LIN {X 0,Y 185.568,Z 561.36,A -85,B 0,C 180,E1 -22347.032,E2 -22347.032} C_VEL
LIN {X 0,Y 185.587,Z 561.366,A -85,B 0,C 180,E1 -22349.493,E2 -22349.493} C_VEL
LIN {X 0,Y 185.509,Z 561.379,A -85,B 0,C 180,E1 -22354.631,E2 -22354.631} C_VEL
LIN {X 0,Y 185.515,Z 561.377,A -85,B 0,C 180,E1 -22357.312,E2 -22357.312} C_VEL
LIN {X 0,Y 185.48,Z 561.382,A -85,B 0,C 180,E1 -22360.724,E2 -22360.724} C_VEL
LIN {X 0,Y 185.468,Z 561.376,A -85,B 0,C 180,E1 -22366.054,E2 -22366.054} C_VEL
LIN {X 0,Y 185.531,Z 561.532,A -85,B 0,C 180,E1 -22368.005,E2 -22368.005} C_VEL
LIN {X 0,Y 186.738,Z 566.432,A -85,B 0,C 180,E1 -22370.786,E2 -22370.786} C_VEL
LIN {X 0,Y 194.108,Z 583.862,A -85,B 0,C 180,E1 -22372.91,E2 -22372.91} C_VEL
LIN {X 0,Y 201.823,Z 604.433,A -85,B 0,C 180,E1 -22375.045,E2 -22375.045} C_VEL
LIN {X 0,Y 204.097,Z 623.143,A -85,B 0,C 180,E1 -22376.201,E2 -22376.201} C_VEL
LIN {X 0,Y 201.981,Z 663.7,A -85,B 0,C 180,E1 -22377.733,E2 -22377.733} C_VEL
LIN {X 0,Y 201.059,Z 669.51,A -85,B 0,C 180,E1 -22377.882,E2 -22377.882} C_VEL
LIN {X 0,Y 197.67,Z 678.837,A -85,B 0,C 180,E1 -22378.008,E2 -22378.008} C_VEL
LIN {X 0,Y 194.055,Z 688.023,A -85,B 0,C 180,E1 -22378.33,E2 -22378.33} C_VEL
LIN {X 0,Y 192.763,Z 693.612,A -85,B 0,C 180,E1 -22378.765,E2 -22378.765} C_VEL
LIN {X 0,Y 191.04,Z 704.06,A -85,B 0,C 180,E1 -22379.915,E2 -22379.915} C_VEL
LIN {X 0,Y 188.782,Z 716.056,A -85,B 0,C 180,E1 -22381.66,E2 -22381.66} C_VEL
LIN {X 0,Y 186.405,Z 726.819,A -85,B 0,C 180,E1 -22383.701,E2 -22383.701} C_VEL
LIN {X 0,Y 184.002,Z 736.963,A -85,B 0,C 180,E1 -22386.144,E2 -22386.144} C_VEL
LIN {X 0,Y 182.039,Z 744.915,A -85,B 0,C 180,E1 -22388.517,E2 -22388.517} C_VEL
LIN {X 0,Y 179.866,Z 753.724,A -85,B 0,C 180,E1 -22391.782,E2 -22391.782} C_VEL
LIN {X 0,Y 178.072,Z 760.784,A -85,B 0,C 180,E1 -22395.132,E2 -22395.132} C_VEL
LIN {X 0,Y 176.994,Z 766.43,A -85,B 0,C 180,E1 -22398.545,E2 -22398.545} C_VEL
LIN {X 0,Y 176.336,Z 770.82,A -85,B 0,C 180,E1 -22401.978,E2 -22401.978} C_VEL
LIN {X 0,Y 176.06,Z 774.084,A -85,B 0,C 180,E1 -22405.418,E2 -22405.418} C_VEL
LIN {X 0,Y 176.025,Z 775.685,A -85,B 0,C 180,E1 -22407.709,E2 -22407.709} C_VEL
LIN {X 0,Y 176.156,Z 776.867,A -85,B 0,C 180,E1 -22409.997,E2 -22409.997} C_VEL
LIN {X 0,Y 175.973,Z 777.736,A -85,B 0,C 180,E1 -22413.172,E2 -22413.172} C_VEL
LIN {X 0,Y 176.142,Z 777.8,A -85,B 0,C 180,E1 -22416.871,E2 -22416.871} C_VEL
LIN {X 0,Y 176.481,Z 777.341,A -85,B 0,C 180,E1 -22419.162,E2 -22419.162} C_VEL
LIN {X 0,Y 177.065,Z 776.47,A -85,B 0,C 180,E1 -22421.443,E2 -22421.443} C_VEL
LIN {X 0,Y 178.915,Z 773.51,A -85,B 0,C 180,E1 -22425.957,E2 -22425.957} C_VEL
LIN {X 0,Y 181.172,Z 770.182,A -85,B 0,C 180,E1 -22429.249,E2 -22429.249} C_VEL
LIN {X 0,Y 183.99,Z 765.836,A -85,B 0,C 180,E1 -22432.453,E2 -22432.453} C_VEL
LIN {X 0,Y 187.769,Z 759.389,A -85,B 0,C 180,E1 -22436.063,E2 -22436.063} C_VEL
LIN {X 0,Y 191.749,Z 752.298,A -85,B 0,C 180,E1 -22439.051,E2 -22439.051} C_VEL
LIN {X 0,Y 196.292,Z 743.558,A -85,B 0,C 180,E1 -22441.874,E2 -22441.874} C_VEL
LIN {X 0,Y 200.452,Z 734.678,A -85,B 0,C 180,E1 -22444.119,E2 -22444.119} C_VEL
LIN {X 0,Y 204.501,Z 725.05,A -85,B 0,C 180,E1 -22446.049,E2 -22446.049} C_VEL
LIN {X 0,Y 208.379,Z 714.565,A -85,B 0,C 180,E1 -22447.68,E2 -22447.68} C_VEL
LIN {X 0,Y 211.849,Z 703.058,A -85,B 0,C 180,E1 -22449.07,E2 -22449.07} C_VEL
LIN {X 0,Y 215.033,Z 690.143,A -85,B 0,C 180,E1 -22450.199,E2 -22450.199} C_VEL
LIN {X 0,Y 217.375,Z 677.531,A -85,B 0,C 180,E1 -22450.945,E2 -22450.945} C_VEL
LIN {X 0,Y 219.026,Z 660.991,A -85,B 0,C 180,E1 -22451.617,E2 -22451.617} C_VEL
LIN {X 0,Y 221.568,Z 630.722,A -85,B 0,C 180,E1 -22452.671,E2 -22452.671} C_VEL
LIN {X 0,Y 217.435,Z 619.879,A -85,B 0,C 180,E1 -22454.973,E2 -22454.973} C_VEL
LIN {X 0,Y 213.68,Z 611.836,A -85,B 0,C 180,E1 -22457.185,E2 -22457.185} C_VEL
LIN {X 0,Y 210.021,Z 604.877,A -85,B 0,C 180,E1 -22459.582,E2 -22459.582} C_VEL
LIN {X 0,Y 207.231,Z 599.872,A -85,B 0,C 180,E1 -22461.655,E2 -22461.655} C_VEL
LIN {X 0,Y 204.208,Z 594.895,A -85,B 0,C 180,E1 -22464.191,E2 -22464.191} C_VEL
LIN {X 0,Y 201.243,Z 589.954,A -85,B 0,C 180,E1 -22467.293,E2 -22467.293} C_VEL
LIN {X 0,Y 197.036,Z 583.326,A -85,B 0,C 180,E1 -22474.09,E2 -22474.09} C_VEL
LIN {X 0,Y 195.819,Z 581.983,A -85,B 0,C 180,E1 -22478.966,E2 -22478.966} C_VEL
LIN {X 0,Y 196.149,Z 581.812,A -85,B 0,C 180,E1 -22483.342,E2 -22483.342} C_VEL
LIN {X 0,Y 196.858,Z 582.371,A -85,B 0,C 180,E1 -22485.725,E2 -22485.725} C_VEL
LIN {X 0,Y 200.195,Z 586.287,A -85,B 0,C 180,E1 -22491.576,E2 -22491.576} C_VEL
LIN {X 0,Y 201.072,Z 587.621,A -85,B 0,C 180,E1 -22492.72,E2 -22492.72} C_VEL
LIN {X 0,Y 203.233,Z 590.314,A -85,B 0,C 180,E1 -22494.976,E2 -22494.976} C_VEL
LIN {X 0,Y 205.193,Z 592.528,A -85,B 0,C 180,E1 -22496.747,E2 -22496.747} C_VEL
LIN {X 0,Y 208.099,Z 597.214,A -85,B 0,C 180,E1 -22499.109,E2 -22499.109} C_VEL
LIN {X 0,Y 212.123,Z 603.731,A -85,B 0,C 180,E1 -22501.898,E2 -22501.898} C_VEL
LIN {X 0,Y 215.695,Z 610.557,A -85,B 0,C 180,E1 -22504.13,E2 -22504.13} C_VEL
LIN {X 0,Y 219.734,Z 618.887,A -85,B 0,C 180,E1 -22506.363,E2 -22506.363} C_VEL
LIN {X 0,Y 221.96,Z 624.2,A -85,B 0,C 180,E1 -22507.553,E2 -22507.553} C_VEL
LIN {X 0,Y 218.205,Z 667.202,A -85,B 0,C 180,E1 -22509.106,E2 -22509.106} C_VEL
LIN {X 0,Y 216.063,Z 680.58,A -85,B 0,C 180,E1 -22509.884,E2 -22509.884} C_VEL
LIN {X 0,Y 213.239,Z 693.467,A -85,B 0,C 180,E1 -22511.023,E2 -22511.023} C_VEL
LIN {X 0,Y 209.684,Z 705.782,A -85,B 0,C 180,E1 -22512.497,E2 -22512.497} C_VEL
LIN {X 0,Y 205.726,Z 717.054,A -85,B 0,C 180,E1 -22514.286,E2 -22514.286} C_VEL
LIN {X 0,Y 201.323,Z 727.735,A -85,B 0,C 180,E1 -22516.523,E2 -22516.523} C_VEL
LIN {X 0,Y 196.767,Z 737.303,A -85,B 0,C 180,E1 -22519.085,E2 -22519.085} C_VEL
LIN {X 0,Y 192.653,Z 744.988,A -85,B 0,C 180,E1 -22521.747,E2 -22521.747} C_VEL
LIN {X 0,Y 188.409,Z 752.132,A -85,B 0,C 180,E1 -22524.957,E2 -22524.957} C_VEL
LIN {X 0,Y 185.285,Z 757.04,A -85,B 0,C 180,E1 -22527.832,E2 -22527.832} C_VEL
LIN {X 0,Y 181.829,Z 762.034,A -85,B 0,C 180,E1 -22531.758,E2 -22531.758} C_VEL
LIN {X 0,Y 179.072,Z 765.618,A -85,B 0,C 180,E1 -22536.063,E2 -22536.063} C_VEL
LIN {X 0,Y 177.63,Z 767.253,A -85,B 0,C 180,E1 -22539.274,E2 -22539.274} C_VEL
LIN {X 0,Y 176.554,Z 768.081,A -85,B 0,C 180,E1 -22542.585,E2 -22542.585} C_VEL
LIN {X 0,Y 175.722,Z 767.804,A -85,B 0,C 180,E1 -22547.168,E2 -22547.168} C_VEL
LIN {X 0,Y 175.569,Z 766.792,A -85,B 0,C 180,E1 -22550.177,E2 -22550.177} C_VEL
LIN {X 0,Y 175.829,Z 763.978,A -85,B 0,C 180,E1 -22554.584,E2 -22554.584} C_VEL
LIN {X 0,Y 176.439,Z 760.818,A -85,B 0,C 180,E1 -22557.876,E2 -22557.876} C_VEL
LIN {X 0,Y 177.436,Z 755.952,A -85,B 0,C 180,E1 -22561.625,E2 -22561.625} C_VEL
LIN {X 0,Y 178.923,Z 749.619,A -85,B 0,C 180,E1 -22565.33,E2 -22565.33} C_VEL
LIN {X 0,Y 180.865,Z 741.806,A -85,B 0,C 180,E1 -22568.838,E2 -22568.838} C_VEL
LIN {X 0,Y 182.779,Z 734.376,A -85,B 0,C 180,E1 -22571.509,E2 -22571.509} C_VEL
LIN {X 0,Y 185.173,Z 724.662,A -85,B 0,C 180,E1 -22574.326,E2 -22574.326} C_VEL
LIN {X 0,Y 187.688,Z 713.78,A -85,B 0,C 180,E1 -22576.793,E2 -22576.793} C_VEL
LIN {X 0,Y 189.969,Z 702.456,A -85,B 0,C 180,E1 -22578.804,E2 -22578.804} C_VEL
LIN {X 0,Y 192.049,Z 690.439,A -85,B 0,C 180,E1 -22580.444,E2 -22580.444} C_VEL
LIN {X 0,Y 193.837,Z 676.765,A -85,B 0,C 180,E1 -22581.793,E2 -22581.793} C_VEL
LIN {X 0,Y 195.137,Z 663.168,A -85,B 0,C 180,E1 -22582.682,E2 -22582.682} C_VEL
LIN {X 0,Y 198.281,Z 606.848,A -85,B 0,C 180,E1 -22584.891,E2 -22584.891} C_VEL
LIN {X 0,Y 189.965,Z 584.27,A -85,B 0,C 180,E1 -22587.286,E2 -22587.286} C_VEL
LIN {X 0,Y 179.493,Z 563.052,A -85,B 0,C 180,E1 -22590.249,E2 -22590.249} C_VEL
LIN {X 0,Y 179.298,Z 562.148,A -85,B 0,C 180,E1 -22590.424,E2 -22590.424} C_VEL
LIN {X 0,Y 178.927,Z 562.19,A -85,B 0,C 180,E1 -22596.77,E2 -22596.77} C_VEL
LIN {X 0,Y 178.86,Z 562.199,A -85,B 0,C 180,E1 -22600.794,E2 -22600.794} C_VEL
LIN {X 0,Y 178.667,Z 562.228,A -85,B 0,C 180,E1 -22605.986,E2 -22605.986} C_VEL
LIN {X 0,Y 178.624,Z 562.227,A -85,B 0,C 180,E1 -22609.219,E2 -22609.219} C_VEL
LIN {X 0,Y 178.536,Z 562.233,A -85,B 0,C 180,E1 -22615.127,E2 -22615.127} C_VEL
LIN {X 0,Y 178.479,Z 562.25,A -85,B 0,C 180,E1 -22620.794,E2 -22620.794} C_VEL
LIN {X 0,Y 178.486,Z 562.25,A -85,B 0,C 180,E1 -22624.222,E2 -22624.222} C_VEL
LIN {X 0,Y 178.399,Z 562.257,A -85,B 0,C 180,E1 -22629.077,E2 -22629.077} C_VEL
LIN {X 0,Y 178.402,Z 562.255,A -85,B 0,C 180,E1 -22632.048,E2 -22632.048} C_VEL
LIN {X 0,Y 178.403,Z 562.263,A -85,B 0,C 180,E1 -22635.165,E2 -22635.165} C_VEL
LIN {X 0,Y 178.408,Z 562.255,A -85,B 0,C 180,E1 -22638.462,E2 -22638.462} C_VEL
LIN {X 0,Y 178.428,Z 562.257,A -85,B 0,C 180,E1 -22643.786,E2 -22643.786} C_VEL
LIN {X 0,Y 178.493,Z 562.25,A -85,B 0,C 180,E1 -22646.55,E2 -22646.55} C_VEL
LIN {X 0,Y 178.529,Z 562.232,A -85,B 0,C 180,E1 -22650.009,E2 -22650.009} C_VEL
LIN {X 0,Y 178.527,Z 562.242,A -85,B 0,C 180,E1 -22654.888,E2 -22654.888} C_VEL
LIN {X 0,Y 178.617,Z 562.226,A -85,B 0,C 180,E1 -22660.799,E2 -22660.799} C_VEL
LIN {X 0,Y 178.659,Z 562.228,A -85,B 0,C 180,E1 -22666.349,E2 -22666.349} C_VEL
LIN {X 0,Y 178.92,Z 562.192,A -85,B 0,C 180,E1 -22670.961,E2 -22670.961} C_VEL
LIN {X 0,Y 179.161,Z 562.167,A -85,B 0,C 180,E1 -22677.753,E2 -22677.753} C_VEL
LIN {X 0,Y 179.379,Z 562.14,A -85,B 0,C 180,E1 -22680.001,E2 -22680.001} C_VEL
LIN {X 0,Y 178.882,Z 562.19,A -85,B 0,C 180,E1 -22684.508,E2 -22684.508} C_VEL
LIN {X 0,Y 178.988,Z 562.189,A -85,B 0,C 180,E1 -22689.037,E2 -22689.037} C_VEL
LIN {X 0,Y 178.676,Z 562.217,A -85,B 0,C 180,E1 -22693.652,E2 -22693.652} C_VEL
LIN {X 0,Y 178.632,Z 562.232,A -85,B 0,C 180,E1 -22699.215,E2 -22699.215} C_VEL
LIN {X 0,Y 178.53,Z 562.217,A -85,B 0,C 180,E1 -22705.114,E2 -22705.114} C_VEL
LIN {X 0,Y 178.531,Z 562.247,A -85,B 0,C 180,E1 -22709.992,E2 -22709.992} C_VEL
LIN {X 0,Y 178.494,Z 562.254,A -85,B 0,C 180,E1 -22714.218,E2 -22714.218} C_VEL
LIN {X 0,Y 178.405,Z 562.262,A -85,B 0,C 180,E1 -22719.073,E2 -22719.073} C_VEL
LIN {X 0,Y 178.407,Z 562.261,A -85,B 0,C 180,E1 -22722.044,E2 -22722.044} C_VEL
LIN {X 0,Y 178.453,Z 562.293,A -85,B 0,C 180,E1 -22727.084,E2 -22727.084} C_VEL
LIN {X 0,Y 179.461,Z 566.426,A -85,B 0,C 180,E1 -22729.464,E2 -22729.464} C_VEL
LIN {X 0,Y 187.25,Z 584.258,A -85,B 0,C 180,E1 -22731.8,E2 -22731.8} C_VEL
LIN {X 0,Y 195.637,Z 606.702,A -85,B 0,C 180,E1 -22734.246,E2 -22734.246} C_VEL
LIN {X 0,Y 197.643,Z 623.334,A -85,B 0,C 180,E1 -22735.32,E2 -22735.32} C_VEL
LIN {X 0,Y 194.819,Z 675.043,A -85,B 0,C 180,E1 -22737.391,E2 -22737.391} C_VEL
LIN {X 0,Y 193.484,Z 687.523,A -85,B 0,C 180,E1 -22738.215,E2 -22738.215} C_VEL
LIN {X 0,Y 192.763,Z 693.612,A -85,B 0,C 180,E1 -22738.765,E2 -22738.765} C_VEL
LIN {X 0,Y 191.927,Z 697.302,A -85,B 0,C 180,E1 -22739.099,E2 -22739.099} C_VEL
LIN {X 0,Y 188.874,Z 704.35,A -85,B 0,C 180,E1 -22739.701,E2 -22739.701} C_VEL
LIN {X 0,Y 182.587,Z 716.046,A -85,B 0,C 180,E1 -22740.989,E2 -22740.989} C_VEL
LIN {X 0,Y 180.955,Z 721.015,A -85,B 0,C 180,E1 -22741.842,E2 -22741.842} C_VEL
LIN {X 0,Y 178.322,Z 732.128,A -85,B 0,C 180,E1 -22744.305,E2 -22744.305} C_VEL
LIN {X 0,Y 175.955,Z 741.248,A -85,B 0,C 180,E1 -22746.853,E2 -22746.853} C_VEL
LIN {X 0,Y 174.196,Z 748.419,A -85,B 0,C 180,E1 -22749.324,E2 -22749.324} C_VEL
LIN {X 0,Y 172.095,Z 756.546,A -85,B 0,C 180,E1 -22752.775,E2 -22752.775} C_VEL
LIN {X 0,Y 170.705,Z 762.018,A -85,B 0,C 180,E1 -22755.695,E2 -22755.695} C_VEL
LIN {X 0,Y 169.725,Z 767.371,A -85,B 0,C 180,E1 -22759.258,E2 -22759.258} C_VEL
LIN {X 0,Y 169.157,Z 771.486,A -85,B 0,C 180,E1 -22762.837,E2 -22762.837} C_VEL
LIN {X 0,Y 168.933,Z 774.775,A -85,B 0,C 180,E1 -22766.833,E2 -22766.833} C_VEL
LIN {X 0,Y 169.06,Z 776.481,A -85,B 0,C 180,E1 -22769.997,E2 -22769.997} C_VEL
LIN {X 0,Y 168.894,Z 777.381,A -85,B 0,C 180,E1 -22772.918,E2 -22772.918} C_VEL
LIN {X 0,Y 169.095,Z 777.617,A -85,B 0,C 180,E1 -22777.159,E2 -22777.159} C_VEL
LIN {X 0,Y 170.09,Z 776.42,A -85,B 0,C 180,E1 -22781.919,E2 -22781.919} C_VEL
LIN {X 0,Y 170.973,Z 775.213,A -85,B 0,C 180,E1 -22784.275,E2 -22784.275} C_VEL
LIN {X 0,Y 172.793,Z 772.668,A -85,B 0,C 180,E1 -22787.757,E2 -22787.757} C_VEL
LIN {X 0,Y 175.426,Z 769.138,A -85,B 0,C 180,E1 -22791.131,E2 -22791.131} C_VEL
LIN {X 0,Y 178.531,Z 764.559,A -85,B 0,C 180,E1 -22794.411,E2 -22794.411} C_VEL
LIN {X 0,Y 182.074,Z 758.817,A -85,B 0,C 180,E1 -22797.59,E2 -22797.59} C_VEL
LIN {X 0,Y 186.418,Z 751.681,A -85,B 0,C 180,E1 -22800.59,E2 -22800.59} C_VEL
LIN {X 0,Y 191.197,Z 742.922,A -85,B 0,C 180,E1 -22803.457,E2 -22803.457} C_VEL
LIN {X 0,Y 196.066,Z 733.037,A -85,B 0,C 180,E1 -22805.938,E2 -22805.938} C_VEL
LIN {X 0,Y 200.368,Z 723.04,A -85,B 0,C 180,E1 -22807.862,E2 -22807.862} C_VEL
LIN {X 0,Y 204.954,Z 710.562,A -85,B 0,C 180,E1 -22809.688,E2 -22809.688} C_VEL
LIN {X 0,Y 208.439,Z 698.994,A -85,B 0,C 180,E1 -22810.944,E2 -22810.944} C_VEL
LIN {X 0,Y 211.524,Z 685.589,A -85,B 0,C 180,E1 -22812.002,E2 -22812.002} C_VEL
LIN {X 0,Y 213.664,Z 672.766,A -85,B 0,C 180,E1 -22812.676,E2 -22812.676} C_VEL
LIN {X 0,Y 217.242,Z 633.882,A -85,B 0,C 180,E1 -22814.062,E2 -22814.062} C_VEL
LIN {X 0,Y 216.224,Z 630.484,A -85,B 0,C 180,E1 -22814.703,E2 -22814.703} C_VEL
LIN {X 0,Y 212.769,Z 621.671,A -85,B 0,C 180,E1 -22816.821,E2 -22816.821} C_VEL
LIN {X 0,Y 209.255,Z 614.22,A -85,B 0,C 180,E1 -22819.158,E2 -22819.158} C_VEL
LIN {X 0,Y 206.872,Z 609.624,A -85,B 0,C 180,E1 -22820.899,E2 -22820.899} C_VEL
LIN {X 0,Y 204.756,Z 605.627,A -85,B 0,C 180,E1 -22822.626,E2 -22822.626} C_VEL
LIN {X 0,Y 202.348,Z 601.388,A -85,B 0,C 180,E1 -22824.819,E2 -22824.819} C_VEL
LIN {X 0,Y 199.536,Z 596.507,A -85,B 0,C 180,E1 -22827.922,E2 -22827.922} C_VEL
LIN {X 0,Y 195.806,Z 590.238,A -85,B 0,C 180,E1 -22834.486,E2 -22834.486} C_VEL
LIN {X 0,Y 194.708,Z 588.892,A -85,B 0,C 180,E1 -22839.787,E2 -22839.787} C_VEL
LIN {X 0,Y 195.605,Z 589.104,A -85,B 0,C 180,E1 -22845.166,E2 -22845.166} C_VEL
LIN {X 0,Y 197.777,Z 592.058,A -85,B 0,C 180,E1 -22849.765,E2 -22849.765} C_VEL
LIN {X 0,Y 199.299,Z 593.862,A -85,B 0,C 180,E1 -22851.89,E2 -22851.89} C_VEL
LIN {X 0,Y 201.478,Z 596.956,A -85,B 0,C 180,E1 -22854.398,E2 -22854.398} C_VEL
LIN {X 0,Y 203.206,Z 598.85,A -85,B 0,C 180,E1 -22856.033,E2 -22856.033} C_VEL
LIN {X 0,Y 205.793,Z 603.268,A -85,B 0,C 180,E1 -22858.296,E2 -22858.296} C_VEL
LIN {X 0,Y 209.899,Z 610.214,A -85,B 0,C 180,E1 -22861.33,E2 -22861.33} C_VEL
LIN {X 0,Y 214.835,Z 620.382,A -85,B 0,C 180,E1 -22864.497,E2 -22864.497} C_VEL
LIN {X 0,Y 217.661,Z 627.045,A -85,B 0,C 180,E1 -22866.127,E2 -22866.127} C_VEL
LIN {X 0,Y 213.925,Z 667.397,A -85,B 0,C 180,E1 -22867.603,E2 -22867.603} C_VEL
LIN {X 0,Y 211.844,Z 679.957,A -85,B 0,C 180,E1 -22868.328,E2 -22868.328} C_VEL
LIN {X 0,Y 208.902,Z 692.992,A -85,B 0,C 180,E1 -22869.458,E2 -22869.458} C_VEL
LIN {X 0,Y 205.11,Z 705.704,A -85,B 0,C 180,E1 -22870.974,E2 -22870.974} C_VEL
LIN {X 0,Y 200.968,Z 717.062,A -85,B 0,C 180,E1 -22872.772,E2 -22872.772} C_VEL
LIN {X 0,Y 196.415,Z 727.596,A -85,B 0,C 180,E1 -22874.976,E2 -22874.976} C_VEL
LIN {X 0,Y 191.618,Z 737.127,A -85,B 0,C 180,E1 -22877.533,E2 -22877.533} C_VEL
LIN {X 0,Y 186.674,Z 745.816,A -85,B 0,C 180,E1 -22880.626,E2 -22880.626} C_VEL
LIN {X 0,Y 181.755,Z 753.527,A -85,B 0,C 180,E1 -22884.281,E2 -22884.281} C_VEL
LIN {X 0,Y 178.463,Z 758.249,A -85,B 0,C 180,E1 -22887.277,E2 -22887.277} C_VEL
LIN {X 0,Y 175.677,Z 761.951,A -85,B 0,C 180,E1 -22890.356,E2 -22890.356} C_VEL
LIN {X 0,Y 172.609,Z 765.631,A -85,B 0,C 180,E1 -22894.751,E2 -22894.751} C_VEL
LIN {X 0,Y 170.77,Z 767.512,A -85,B 0,C 180,E1 -22898.567,E2 -22898.567} C_VEL
LIN {X 0,Y 169.657,Z 768.284,A -85,B 0,C 180,E1 -22901.791,E2 -22901.791} C_VEL
LIN {X 0,Y 168.922,Z 768.289,A -85,B 0,C 180,E1 -22905.012,E2 -22905.012} C_VEL
LIN {X 0,Y 168.512,Z 767.446,A -85,B 0,C 180,E1 -22908.65,E2 -22908.65} C_VEL
LIN {X 0,Y 168.516,Z 765.591,A -85,B 0,C 180,E1 -22912.408,E2 -22912.408} C_VEL
LIN {X 0,Y 169.005,Z 762.581,A -85,B 0,C 180,E1 -22916.27,E2 -22916.27} C_VEL
LIN {X 0,Y 169.908,Z 758.132,A -85,B 0,C 180,E1 -22920.298,E2 -22920.298} C_VEL
LIN {X 0,Y 171.117,Z 752.906,A -85,B 0,C 180,E1 -22923.853,E2 -22923.853} C_VEL
LIN {X 0,Y 172.736,Z 746.503,A -85,B 0,C 180,E1 -22927.266,E2 -22927.266} C_VEL
LIN {X 0,Y 174.895,Z 738.452,A -85,B 0,C 180,E1 -22930.643,E2 -22930.643} C_VEL
LIN {X 0,Y 176.954,Z 730.378,A -85,B 0,C 180,E1 -22933.368,E2 -22933.368} C_VEL
LIN {X 0,Y 179.551,Z 720.14,A -85,B 0,C 180,E1 -22936.132,E2 -22936.132} C_VEL
LIN {X 0,Y 181.869,Z 709.949,A -85,B 0,C 180,E1 -22938.298,E2 -22938.298} C_VEL
LIN {X 0,Y 184.186,Z 698.043,A -85,B 0,C 180,E1 -22940.28,E2 -22940.28} C_VEL
LIN {X 0,Y 186.316,Z 685.283,A -85,B 0,C 180,E1 -22941.871,E2 -22941.871} C_VEL
LIN {X 0,Y 187.915,Z 671.4,A -85,B 0,C 180,E1 -22943.089,E2 -22943.089} C_VEL
LIN {X 0,Y 189.03,Z 658.7,A -85,B 0,C 180,E1 -22943.782,E2 -22943.782} C_VEL
LIN {X 0,Y 191.852,Z 608.295,A -85,B 0,C 180,E1 -22945.802,E2 -22945.802} C_VEL
LIN {X 0,Y 184.175,Z 587.474,A -85,B 0,C 180,E1 -22948.1,E2 -22948.1} C_VEL
LIN {X 0,Y 174.053,Z 566.979,A -85,B 0,C 180,E1 -22951.122,E2 -22951.122} C_VEL
LIN {X 0,Y 172.534,Z 564.575,A -85,B 0,C 180,E1 -22951.574,E2 -22951.574} C_VEL
LIN {X 0,Y 172.151,Z 563.038,A -85,B 0,C 180,E1 -22951.758,E2 -22951.758} C_VEL
LIN {X 0,Y 171.891,Z 563.068,A -85,B 0,C 180,E1 -22957.049,E2 -22957.049} C_VEL
LIN {X 0,Y 171.793,Z 563.078,A -85,B 0,C 180,E1 -22960.945,E2 -22960.945} C_VEL
LIN {X 0,Y 171.587,Z 563.112,A -85,B 0,C 180,E1 -22966.665,E2 -22966.665} C_VEL
LIN {X 0,Y 171.545,Z 563.107,A -85,B 0,C 180,E1 -22969.565,E2 -22969.565} C_VEL
LIN {X 0,Y 171.47,Z 563.117,A -85,B 0,C 180,E1 -22975.619,E2 -22975.619} C_VEL
LIN {X 0,Y 171.442,Z 563.128,A -85,B 0,C 180,E1 -22980.589,E2 -22980.589} C_VEL
LIN {X 0,Y 171.395,Z 563.135,A -85,B 0,C 180,E1 -22985.038,E2 -22985.038} C_VEL
LIN {X 0,Y 171.361,Z 563.135,A -85,B 0,C 180,E1 -22988.811,E2 -22988.811} C_VEL
LIN {X 0,Y 171.33,Z 563.142,A -85,B 0,C 180,E1 -22994.218,E2 -22994.218} C_VEL
LIN {X 0,Y 171.34,Z 563.13,A -85,B 0,C 180,E1 -22998.985,E2 -22998.985} C_VEL
LIN {X 0,Y 171.392,Z 563.125,A -85,B 0,C 180,E1 -23002.044,E2 -23002.044} C_VEL
LIN {X 0,Y 171.404,Z 563.133,A -85,B 0,C 180,E1 -23005.095,E2 -23005.095} C_VEL
LIN {X 0,Y 171.455,Z 563.111,A -85,B 0,C 180,E1 -23010.537,E2 -23010.537} C_VEL
LIN {X 0,Y 171.451,Z 563.128,A -85,B 0,C 180,E1 -23015.802,E2 -23015.802} C_VEL
LIN {X 0,Y 171.573,Z 563.101,A -85,B 0,C 180,E1 -23020.872,E2 -23020.872} C_VEL
LIN {X 0,Y 171.576,Z 563.107,A -85,B 0,C 180,E1 -23025.774,E2 -23025.774} C_VEL
LIN {X 0,Y 171.857,Z 563.072,A -85,B 0,C 180,E1 -23030.587,E2 -23030.587} C_VEL
LIN {X 0,Y 171.823,Z 563.07,A -85,B 0,C 180,E1 -23035.309,E2 -23035.309} C_VEL
LIN {X 0,Y 172.342,Z 563.016,A -85,B 0,C 180,E1 -23040.001,E2 -23040.001} C_VEL
LIN {X 0,Y 171.832,Z 563.068,A -85,B 0,C 180,E1 -23044.693,E2 -23044.693} C_VEL
LIN {X 0,Y 171.914,Z 563.071,A -85,B 0,C 180,E1 -23049.413,E2 -23049.413} C_VEL
LIN {X 0,Y 171.592,Z 563.103,A -85,B 0,C 180,E1 -23054.227,E2 -23054.227} C_VEL
LIN {X 0,Y 171.552,Z 563.111,A -85,B 0,C 180,E1 -23059.559,E2 -23059.559} C_VEL
LIN {X 0,Y 171.468,Z 563.099,A -85,B 0,C 180,E1 -23065.608,E2 -23065.608} C_VEL
LIN {X 0,Y 171.45,Z 563.127,A -85,B 0,C 180,E1 -23070.585,E2 -23070.585} C_VEL
LIN {X 0,Y 171.402,Z 563.135,A -85,B 0,C 180,E1 -23075.034,E2 -23075.034} C_VEL
LIN {X 0,Y 171.367,Z 563.139,A -85,B 0,C 180,E1 -23078.806,E2 -23078.806} C_VEL
LIN {X 0,Y 171.33,Z 563.141,A -85,B 0,C 180,E1 -23084.216,E2 -23084.216} C_VEL
LIN {X 0,Y 171.39,Z 563.23,A -85,B 0,C 180,E1 -23086.198,E2 -23086.198} C_VEL
LIN {X 0,Y 172.119,Z 566.116,A -85,B 0,C 180,E1 -23087.954,E2 -23087.954} C_VEL
LIN {X 0,Y 179.955,Z 583.631,A -85,B 0,C 180,E1 -23090.481,E2 -23090.481} C_VEL
LIN {X 0,Y 188.217,Z 605.357,A -85,B 0,C 180,E1 -23093.012,E2 -23093.012} C_VEL
LIN {X 0,Y 189.562,Z 609.48,A -85,B 0,C 180,E1 -23093.431,E2 -23093.431} C_VEL
LIN {X 0,Y 191.264,Z 624.539,A -85,B 0,C 180,E1 -23094.434,E2 -23094.434} C_VEL
LIN {X 0,Y 188.36,Z 675.155,A -85,B 0,C 180,E1 -23096.526,E2 -23096.526} C_VEL
LIN {X 0,Y 186.87,Z 688.248,A -85,B 0,C 180,E1 -23097.43,E2 -23097.43} C_VEL
LIN {X 0,Y 185.022,Z 700.485,A -85,B 0,C 180,E1 -23098.67,E2 -23098.67} C_VEL
LIN {X 0,Y 183.16,Z 710.788,A -85,B 0,C 180,E1 -23100.075,E2 -23100.075} C_VEL
LIN {X 0,Y 180.955,Z 721.015,A -85,B 0,C 180,E1 -23101.842,E2 -23101.842} C_VEL
LIN {X 0,Y 179.983,Z 724.29,A -85,B 0,C 180,E1 -23102.469,E2 -23102.469} C_VEL
LIN {X 0,Y 176.597,Z 730.43,A -85,B 0,C 180,E1 -23103.666,E2 -23103.666} C_VEL
LIN {X 0,Y 169.868,Z 740.256,A -85,B 0,C 180,E1 -23106.066,E2 -23106.066} C_VEL
LIN {X 0,Y 168.26,Z 744.347,A -85,B 0,C 180,E1 -23107.405,E2 -23107.405} C_VEL
LIN {X 0,Y 165.967,Z 752.979,A -85,B 0,C 180,E1 -23110.838,E2 -23110.838} C_VEL
LIN {X 0,Y 164.044,Z 760.117,A -85,B 0,C 180,E1 -23114.465,E2 -23114.465} C_VEL
LIN {X 0,Y 162.731,Z 766.632,A -85,B 0,C 180,E1 -23118.79,E2 -23118.79} C_VEL
LIN {X 0,Y 162.115,Z 770.872,A -85,B 0,C 180,E1 -23122.524,E2 -23122.524} C_VEL
LIN {X 0,Y 161.927,Z 773.093,A -85,B 0,C 180,E1 -23125.017,E2 -23125.017} C_VEL
LIN {X 0,Y 161.869,Z 774.804,A -85,B 0,C 180,E1 -23127.508,E2 -23127.508} C_VEL
LIN {X 0,Y 161.966,Z 776.09,A -85,B 0,C 180,E1 -23129.996,E2 -23129.996} C_VEL
LIN {X 0,Y 161.8,Z 776.951,A -85,B 0,C 180,E1 -23132.486,E2 -23132.486} C_VEL
LIN {X 0,Y 161.852,Z 777.407,A -85,B 0,C 180,E1 -23134.979,E2 -23134.979} C_VEL
LIN {X 0,Y 162.442,Z 777.08,A -85,B 0,C 180,E1 -23139.962,E2 -23139.962} C_VEL
LIN {X 0,Y 164.079,Z 775.243,A -85,B 0,C 180,E1 -23144.888,E2 -23144.888} C_VEL
LIN {X 0,Y 165.257,Z 773.706,A -85,B 0,C 180,E1 -23147.315,E2 -23147.315} C_VEL
LIN {X 0,Y 167.81,Z 770.634,A -85,B 0,C 180,E1 -23150.85,E2 -23150.85} C_VEL
LIN {X 0,Y 170.935,Z 766.544,A -85,B 0,C 180,E1 -23154.273,E2 -23154.273} C_VEL
LIN {X 0,Y 174.927,Z 760.807,A -85,B 0,C 180,E1 -23157.883,E2 -23157.883} C_VEL
LIN {X 0,Y 179.563,Z 753.708,A -85,B 0,C 180,E1 -23161.234,E2 -23161.234} C_VEL
LIN {X 0,Y 184.5,Z 745.501,A -85,B 0,C 180,E1 -23164.18,E2 -23164.18} C_VEL
LIN {X 0,Y 189.053,Z 737.153,A -85,B 0,C 180,E1 -23166.494,E2 -23166.494} C_VEL
LIN {X 0,Y 193.895,Z 726.981,A -85,B 0,C 180,E1 -23168.697,E2 -23168.697} C_VEL
LIN {X 0,Y 198.584,Z 715.696,A -85,B 0,C 180,E1 -23170.56,E2 -23170.56} C_VEL
LIN {X 0,Y 202.371,Z 704.743,A -85,B 0,C 180,E1 -23171.949,E2 -23171.949} C_VEL
LIN {X 0,Y 205.807,Z 692.559,A -85,B 0,C 180,E1 -23173.072,E2 -23173.072} C_VEL
LIN {X 0,Y 208.338,Z 680.87,A -85,B 0,C 180,E1 -23173.837,E2 -23173.837} C_VEL
LIN {X 0,Y 210.238,Z 666.915,A -85,B 0,C 180,E1 -23174.489,E2 -23174.489} C_VEL
LIN {X 0,Y 213.062,Z 636.036,A -85,B 0,C 180,E1 -23175.594,E2 -23175.594} C_VEL
LIN {X 0,Y 209.87,Z 627.208,A -85,B 0,C 180,E1 -23177.744,E2 -23177.744} C_VEL
LIN {X 0,Y 206.686,Z 620.131,A -85,B 0,C 180,E1 -23179.993,E2 -23179.993} C_VEL
LIN {X 0,Y 203.158,Z 612.726,A -85,B 0,C 180,E1 -23182.915,E2 -23182.915} C_VEL
LIN {X 0,Y 200.413,Z 607.725,A -85,B 0,C 180,E1 -23185.562,E2 -23185.562} C_VEL
LIN {X 0,Y 197.799,Z 602.988,A -85,B 0,C 180,E1 -23188.691,E2 -23188.691} C_VEL
LIN {X 0,Y 194.53,Z 597.085,A -85,B 0,C 180,E1 -23195.004,E2 -23195.004} C_VEL
LIN {X 0,Y 193.645,Z 595.824,A -85,B 0,C 180,E1 -23200.659,E2 -23200.659} C_VEL
LIN {X 0,Y 194.428,Z 596.053,A -85,B 0,C 180,E1 -23204.878,E2 -23204.878} C_VEL
LIN {X 0,Y 196.385,Z 598.879,A -85,B 0,C 180,E1 -23209.325,E2 -23209.325} C_VEL
LIN {X 0,Y 197.71,Z 600.414,A -85,B 0,C 180,E1 -23211.259,E2 -23211.259} C_VEL
LIN {X 0,Y 199.667,Z 603.486,A -85,B 0,C 180,E1 -23213.728,E2 -23213.728} C_VEL
LIN {X 0,Y 201.291,Z 605.224,A -85,B 0,C 180,E1 -23215.331,E2 -23215.331} C_VEL
LIN {X 0,Y 203.615,Z 609.484,A -85,B 0,C 180,E1 -23217.545,E2 -23217.545} C_VEL
LIN {X 0,Y 207.515,Z 616.508,A -85,B 0,C 180,E1 -23220.637,E2 -23220.637} C_VEL
LIN {X 0,Y 211.754,Z 625.735,A -85,B 0,C 180,E1 -23223.537,E2 -23223.537} C_VEL
LIN {X 0,Y 213.51,Z 630.019,A -85,B 0,C 180,E1 -23224.655,E2 -23224.655} C_VEL
LIN {X 0,Y 209.9,Z 667.334,A -85,B 0,C 180,E1 -23226.019,E2 -23226.019} C_VEL
LIN {X 0,Y 207.655,Z 680.352,A -85,B 0,C 180,E1 -23226.761,E2 -23226.761} C_VEL
LIN {X 0,Y 204.57,Z 693.413,A -85,B 0,C 180,E1 -23227.898,E2 -23227.898} C_VEL
LIN {X 0,Y 201.061,Z 704.804,A -85,B 0,C 180,E1 -23229.253,E2 -23229.253} C_VEL
LIN {X 0,Y 196.85,Z 715.9,A -85,B 0,C 180,E1 -23230.963,E2 -23230.963} C_VEL
LIN {X 0,Y 192.573,Z 725.607,A -85,B 0,C 180,E1 -23232.913,E2 -23232.913} C_VEL
LIN {X 0,Y 188.025,Z 734.495,A -85,B 0,C 180,E1 -23235.167,E2 -23235.167} C_VEL
LIN {X 0,Y 183.234,Z 742.781,A -85,B 0,C 180,E1 -23237.868,E2 -23237.868} C_VEL
LIN {X 0,Y 178.922,Z 749.524,A -85,B 0,C 180,E1 -23240.701,E2 -23240.701} C_VEL
LIN {X 0,Y 174.982,Z 755.066,A -85,B 0,C 180,E1 -23243.679,E2 -23243.679} C_VEL
LIN {X 0,Y 171.541,Z 759.52,A -85,B 0,C 180,E1 -23246.785,E2 -23246.785} C_VEL
LIN {X 0,Y 167.674,Z 764.132,A -85,B 0,C 180,E1 -23251.269,E2 -23251.269} C_VEL
LIN {X 0,Y 166.266,Z 765.645,A -85,B 0,C 180,E1 -23253.332,E2 -23253.332} C_VEL
LIN {X 0,Y 164.37,Z 767.418,A -85,B 0,C 180,E1 -23256.768,E2 -23256.768} C_VEL
LIN {X 0,Y 162.979,Z 768.386,A -85,B 0,C 180,E1 -23260.301,E2 -23260.301} C_VEL
LIN {X 0,Y 162.004,Z 768.543,A -85,B 0,C 180,E1 -23263.954,E2 -23263.954} C_VEL
LIN {X 0,Y 161.462,Z 767.818,A -85,B 0,C 180,E1 -23267.726,E2 -23267.726} C_VEL
LIN {X 0,Y 161.418,Z 765.6,A -85,B 0,C 180,E1 -23272.448,E2 -23272.448} C_VEL
LIN {X 0,Y 162.068,Z 761.844,A -85,B 0,C 180,E1 -23277.181,E2 -23277.181} C_VEL
LIN {X 0,Y 162.906,Z 757.83,A -85,B 0,C 180,E1 -23280.763,E2 -23280.763} C_VEL
LIN {X 0,Y 164.307,Z 752.072,A -85,B 0,C 180,E1 -23284.68,E2 -23284.68} C_VEL
LIN {X 0,Y 166.192,Z 744.867,A -85,B 0,C 180,E1 -23288.485,E2 -23288.485} C_VEL
LIN {X 0,Y 168.356,Z 737.151,A -85,B 0,C 180,E1 -23291.702,E2 -23291.702} C_VEL
LIN {X 0,Y 170.842,Z 727.796,A -85,B 0,C 180,E1 -23294.8,E2 -23294.8} C_VEL
LIN {X 0,Y 173.651,Z 716.703,A -85,B 0,C 180,E1 -23297.669,E2 -23297.669} C_VEL
LIN {X 0,Y 176.228,Z 705.286,A -85,B 0,C 180,E1 -23299.955,E2 -23299.955} C_VEL
LIN {X 0,Y 178.706,Z 692.119,A -85,B 0,C 180,E1 -23301.949,E2 -23301.949} C_VEL
LIN {X 0,Y 180.566,Z 679.605,A -85,B 0,C 180,E1 -23303.333,E2 -23303.333} C_VEL
LIN {X 0,Y 182.015,Z 666.866,A -85,B 0,C 180,E1 -23304.291,E2 -23304.291} C_VEL
LIN {X 0,Y 183.522,Z 643.161,A -85,B 0,C 180,E1 -23305.363,E2 -23305.363} C_VEL
LIN {X 0,Y 185.417,Z 609.703,A -85,B 0,C 180,E1 -23306.752,E2 -23306.752} C_VEL
LIN {X 0,Y 178.628,Z 591.12,A -85,B 0,C 180,E1 -23308.905,E2 -23308.905} C_VEL
LIN {X 0,Y 168.975,Z 571.456,A -85,B 0,C 180,E1 -23311.92,E2 -23311.92} C_VEL
LIN {X 0,Y 165.178,Z 565.112,A -85,B 0,C 180,E1 -23313.128,E2 -23313.128} C_VEL
LIN {X 0,Y 164.908,Z 563.942,A -85,B 0,C 180,E1 -23313.363,E2 -23313.363} C_VEL
LIN {X 0,Y 164.853,Z 563.946,A -85,B 0,C 180,E1 -23317.351,E2 -23317.351} C_VEL
LIN {X 0,Y 164.744,Z 563.953,A -85,B 0,C 180,E1 -23321.139,E2 -23321.139} C_VEL
LIN {X 0,Y 164.507,Z 563.994,A -85,B 0,C 180,E1 -23327.404,E2 -23327.404} C_VEL
LIN {X 0,Y 164.474,Z 563.981,A -85,B 0,C 180,E1 -23329.993,E2 -23329.993} C_VEL
LIN {X 0,Y 164.394,Z 564.003,A -85,B 0,C 180,E1 -23336.137,E2 -23336.137} C_VEL
LIN {X 0,Y 164.376,Z 564.003,A -85,B 0,C 180,E1 -23341.23,E2 -23341.23} C_VEL
LIN {X 0,Y 164.297,Z 564.021,A -85,B 0,C 180,E1 -23346.793,E2 -23346.793} C_VEL
LIN {X 0,Y 164.294,Z 564.008,A -85,B 0,C 180,E1 -23349.919,E2 -23349.919} C_VEL
LIN {X 0,Y 164.283,Z 564.017,A -85,B 0,C 180,E1 -23353.345,E2 -23353.345} C_VEL
LIN {X 0,Y 164.297,Z 564.019,A -85,B 0,C 180,E1 -23356.812,E2 -23356.812} C_VEL
LIN {X 0,Y 164.3,Z 564,A -85,B 0,C 180,E1 -23360.355,E2 -23360.355} C_VEL
LIN {X 0,Y 164.336,Z 564.013,A -85,B 0,C 180,E1 -23364.352,E2 -23364.352} C_VEL
LIN {X 0,Y 164.397,Z 563.997,A -85,B 0,C 180,E1 -23369.138,E2 -23369.138} C_VEL
LIN {X 0,Y 164.413,Z 564,A -85,B 0,C 180,E1 -23374.695,E2 -23374.695} C_VEL
LIN {X 0,Y 164.47,Z 563.988,A -85,B 0,C 180,E1 -23380.074,E2 -23380.074} C_VEL
LIN {X 0,Y 164.506,Z 563.984,A -85,B 0,C 180,E1 -23385.149,E2 -23385.149} C_VEL
LIN {X 0,Y 164.777,Z 563.955,A -85,B 0,C 180,E1 -23390.178,E2 -23390.178} C_VEL
LIN {X 0,Y 164.84,Z 563.936,A -85,B 0,C 180,E1 -23392.653,E2 -23392.653} C_VEL
LIN {X 0,Y 165.056,Z 563.922,A -85,B 0,C 180,E1 -23397.561,E2 -23397.561} C_VEL
LIN {X 0,Y 165.304,Z 563.893,A -85,B 0,C 180,E1 -23400.001,E2 -23400.001} C_VEL
LIN {X 0,Y 164.87,Z 563.946,A -85,B 0,C 180,E1 -23407.348,E2 -23407.348} C_VEL
LIN {X 0,Y 164.76,Z 563.958,A -85,B 0,C 180,E1 -23411.146,E2 -23411.146} C_VEL
LIN {X 0,Y 164.494,Z 563.997,A -85,B 0,C 180,E1 -23417.403,E2 -23417.403} C_VEL
LIN {X 0,Y 164.483,Z 563.987,A -85,B 0,C 180,E1 -23419.989,E2 -23419.989} C_VEL
LIN {X 0,Y 164.395,Z 563.985,A -85,B 0,C 180,E1 -23426.127,E2 -23426.127} C_VEL
LIN {X 0,Y 164.384,Z 564.006,A -85,B 0,C 180,E1 -23431.226,E2 -23431.226} C_VEL
LIN {X 0,Y 164.304,Z 564.019,A -85,B 0,C 180,E1 -23436.788,E2 -23436.788} C_VEL
LIN {X 0,Y 164.3,Z 564.018,A -85,B 0,C 180,E1 -23439.915,E2 -23439.915} C_VEL
LIN {X 0,Y 164.299,Z 564.093,A -85,B 0,C 180,E1 -23445.22,E2 -23445.22} C_VEL
LIN {X 0,Y 164.773,Z 566.021,A -85,B 0,C 180,E1 -23446.367,E2 -23446.367} C_VEL
LIN {X 0,Y 172.1,Z 581.703,A -85,B 0,C 180,E1 -23448.838,E2 -23448.838} C_VEL
LIN {X 0,Y 178.399,Z 597.553,A -85,B 0,C 180,E1 -23450.936,E2 -23450.936} C_VEL
LIN {X 0,Y 183.381,Z 611.315,A -85,B 0,C 180,E1 -23452.524,E2 -23452.524} C_VEL
LIN {X 0,Y 184.92,Z 625.31,A -85,B 0,C 180,E1 -23453.486,E2 -23453.486} C_VEL
LIN {X 0,Y 181.95,Z 674.923,A -85,B 0,C 180,E1 -23455.601,E2 -23455.601} C_VEL
LIN {X 0,Y 180.404,Z 687.987,A -85,B 0,C 180,E1 -23456.528,E2 -23456.528} C_VEL
LIN {X 0,Y 178.582,Z 699.662,A -85,B 0,C 180,E1 -23457.738,E2 -23457.738} C_VEL
LIN {X 0,Y 176.665,Z 710.09,A -85,B 0,C 180,E1 -23459.187,E2 -23459.187} C_VEL
LIN {X 0,Y 174.002,Z 722.001,A -85,B 0,C 180,E1 -23461.335,E2 -23461.335} C_VEL
LIN {X 0,Y 171.39,Z 732.692,A -85,B 0,C 180,E1 -23463.841,E2 -23463.841} C_VEL
LIN {X 0,Y 168.812,Z 741.869,A -85,B 0,C 180,E1 -23466.54,E2 -23466.54} C_VEL
LIN {X 0,Y 168.26,Z 744.347,A -85,B 0,C 180,E1 -23467.405,E2 -23467.405} C_VEL
LIN {X 0,Y 167.369,Z 746.996,A -85,B 0,C 180,E1 -23468.358,E2 -23468.358} C_VEL
LIN {X 0,Y 165.085,Z 750.683,A -85,B 0,C 180,E1 -23469.757,E2 -23469.757} C_VEL
LIN {X 0,Y 158.586,Z 758.209,A -85,B 0,C 180,E1 -23473.238,E2 -23473.238} C_VEL
LIN {X 0,Y 156.764,Z 761.191,A -85,B 0,C 180,E1 -23474.98,E2 -23474.98} C_VEL
LIN {X 0,Y 156.47,Z 762.168,A -85,B 0,C 180,E1 -23475.597,E2 -23475.597} C_VEL
LIN {X 0,Y 155.452,Z 767.498,A -85,B 0,C 180,E1 -23479.578,E2 -23479.578} C_VEL
LIN {X 0,Y 154.909,Z 771.472,A -85,B 0,C 180,E1 -23483.484,E2 -23483.484} C_VEL
LIN {X 0,Y 154.779,Z 774.354,A -85,B 0,C 180,E1 -23487.394,E2 -23487.394} C_VEL
LIN {X 0,Y 154.874,Z 775.692,A -85,B 0,C 180,E1 -23489.996,E2 -23489.996} C_VEL
LIN {X 0,Y 154.719,Z 776.603,A -85,B 0,C 180,E1 -23492.6,E2 -23492.6} C_VEL
LIN {X 0,Y 154.761,Z 777.126,A -85,B 0,C 180,E1 -23495.207,E2 -23495.207} C_VEL
LIN {X 0,Y 154.971,Z 777.25,A -85,B 0,C 180,E1 -23497.816,E2 -23497.816} C_VEL
LIN {X 0,Y 156.186,Z 776.284,A -85,B 0,C 180,E1 -23502.998,E2 -23502.998} C_VEL
LIN {X 0,Y 158.476,Z 773.8,A -85,B 0,C 180,E1 -23508.081,E2 -23508.081} C_VEL
LIN {X 0,Y 161.195,Z 770.842,A -85,B 0,C 180,E1 -23511.748,E2 -23511.748} C_VEL
LIN {X 0,Y 164.48,Z 766.898,A -85,B 0,C 180,E1 -23515.291,E2 -23515.291} C_VEL
LIN {X 0,Y 168.59,Z 761.53,A -85,B 0,C 180,E1 -23518.902,E2 -23518.902} C_VEL
LIN {X 0,Y 173.585,Z 754.435,A -85,B 0,C 180,E1 -23522.439,E2 -23522.439} C_VEL
LIN {X 0,Y 178.729,Z 746.452,A -85,B 0,C 180,E1 -23525.446,E2 -23525.446} C_VEL
LIN {X 0,Y 184.451,Z 736.615,A -85,B 0,C 180,E1 -23528.251,E2 -23528.251} C_VEL
LIN {X 0,Y 189.037,Z 727.541,A -85,B 0,C 180,E1 -23530.234,E2 -23530.234} C_VEL
LIN {X 0,Y 193.901,Z 716.412,A -85,B 0,C 180,E1 -23532.104,E2 -23532.104} C_VEL
LIN {X 0,Y 197.846,Z 705.656,A -85,B 0,C 180,E1 -23533.487,E2 -23533.487} C_VEL
LIN {X 0,Y 201.558,Z 693.267,A -85,B 0,C 180,E1 -23534.663,E2 -23534.663} C_VEL
LIN {X 0,Y 204.334,Z 681.114,A -85,B 0,C 180,E1 -23535.462,E2 -23535.462} C_VEL
LIN {X 0,Y 206.3,Z 667.72,A -85,B 0,C 180,E1 -23536.1,E2 -23536.1} C_VEL
LIN {X 0,Y 209.096,Z 638.868,A -85,B 0,C 180,E1 -23537.148,E2 -23537.148} C_VEL
LIN {X 0,Y 206.519,Z 631.443,A -85,B 0,C 180,E1 -23539.066,E2 -23539.066} C_VEL
LIN {X 0,Y 203.569,Z 624.557,A -85,B 0,C 180,E1 -23541.407,E2 -23541.407} C_VEL
LIN {X 0,Y 200.539,Z 618.09,A -85,B 0,C 180,E1 -23544.144,E2 -23544.144} C_VEL
LIN {X 0,Y 198.456,Z 613.985,A -85,B 0,C 180,E1 -23546.378,E2 -23546.378} C_VEL
LIN {X 0,Y 196.209,Z 609.588,A -85,B 0,C 180,E1 -23549.325,E2 -23549.325} C_VEL
LIN {X 0,Y 193.336,Z 604.018,A -85,B 0,C 180,E1 -23555.329,E2 -23555.329} C_VEL
LIN {X 0,Y 192.594,Z 602.816,A -85,B 0,C 180,E1 -23560.826,E2 -23560.826} C_VEL
LIN {X 0,Y 193.307,Z 603.168,A -85,B 0,C 180,E1 -23564.788,E2 -23564.788} C_VEL
LIN {X 0,Y 196.079,Z 606.852,A -85,B 0,C 180,E1 -23570.516,E2 -23570.516} C_VEL
LIN {X 0,Y 198.124,Z 610.248,A -85,B 0,C 180,E1 -23573.304,E2 -23573.304} C_VEL
LIN {X 0,Y 199.528,Z 611.846,A -85,B 0,C 180,E1 -23574.753,E2 -23574.753} C_VEL
LIN {X 0,Y 201.628,Z 616.015,A -85,B 0,C 180,E1 -23576.921,E2 -23576.921} C_VEL
LIN {X 0,Y 204.968,Z 622.229,A -85,B 0,C 180,E1 -23579.714,E2 -23579.714} C_VEL
LIN {X 0,Y 209.164,Z 631.994,A -85,B 0,C 180,E1 -23582.819,E2 -23582.819} C_VEL
LIN {X 0,Y 209.593,Z 633.135,A -85,B 0,C 180,E1 -23583.121,E2 -23583.121} C_VEL
LIN {X 0,Y 206.032,Z 667.573,A -85,B 0,C 180,E1 -23584.374,E2 -23584.374} C_VEL
LIN {X 0,Y 203.633,Z 680.903,A -85,B 0,C 180,E1 -23585.144,E2 -23585.144} C_VEL
LIN {X 0,Y 200.409,Z 693.828,A -85,B 0,C 180,E1 -23586.275,E2 -23586.275} C_VEL
LIN {X 0,Y 196.332,Z 706.364,A -85,B 0,C 180,E1 -23587.788,E2 -23587.788} C_VEL
LIN {X 0,Y 191.831,Z 717.506,A -85,B 0,C 180,E1 -23589.555,E2 -23589.555} C_VEL
LIN {X 0,Y 186.682,Z 728.237,A -85,B 0,C 180,E1 -23591.83,E2 -23591.83} C_VEL
LIN {X 0,Y 181.406,Z 737.659,A -85,B 0,C 180,E1 -23594.423,E2 -23594.423} C_VEL
LIN {X 0,Y 176.522,Z 745.309,A -85,B 0,C 180,E1 -23597.164,E2 -23597.164} C_VEL
LIN {X 0,Y 172.112,Z 751.624,A -85,B 0,C 180,E1 -23600.097,E2 -23600.097} C_VEL
LIN {X 0,Y 168.11,Z 756.745,A -85,B 0,C 180,E1 -23603.123,E2 -23603.123} C_VEL
LIN {X 0,Y 163.533,Z 762.019,A -85,B 0,C 180,E1 -23607.418,E2 -23607.418} C_VEL
LIN {X 0,Y 160.04,Z 765.635,A -85,B 0,C 180,E1 -23611.799,E2 -23611.799} C_VEL
LIN {X 0,Y 157.322,Z 767.914,A -85,B 0,C 180,E1 -23616.482,E2 -23616.482} C_VEL
LIN {X 0,Y 155.938,Z 768.703,A -85,B 0,C 180,E1 -23619.995,E2 -23619.995} C_VEL
LIN {X 0,Y 155.003,Z 768.738,A -85,B 0,C 180,E1 -23623.499,E2 -23623.499} C_VEL
LIN {X 0,Y 154.421,Z 768.102,A -85,B 0,C 180,E1 -23626.952,E2 -23626.952} C_VEL
LIN {X 0,Y 154.247,Z 766.583,A -85,B 0,C 180,E1 -23630.764,E2 -23630.764} C_VEL
LIN {X 0,Y 154.564,Z 763.892,A -85,B 0,C 180,E1 -23634.928,E2 -23634.928} C_VEL
LIN {X 0,Y 155.418,Z 759.873,A -85,B 0,C 180,E1 -23639.222,E2 -23639.222} C_VEL
LIN {X 0,Y 156.755,Z 754.119,A -85,B 0,C 180,E1 -23643.723,E2 -23643.723} C_VEL
LIN {X 0,Y 158.408,Z 747.948,A -85,B 0,C 180,E1 -23647.433,E2 -23647.433} C_VEL
LIN {X 0,Y 160.389,Z 740.872,A -85,B 0,C 180,E1 -23650.818,E2 -23650.818} C_VEL
LIN {X 0,Y 163.07,Z 731.399,A -85,B 0,C 180,E1 -23654.377,E2 -23654.377} C_VEL
LIN {X 0,Y 165.893,Z 720.959,A -85,B 0,C 180,E1 -23657.442,E2 -23657.442} C_VEL
LIN {X 0,Y 168.456,Z 710.731,A -85,B 0,C 180,E1 -23659.79,E2 -23659.79} C_VEL
LIN {X 0,Y 171.036,Z 698.38,A -85,B 0,C 180,E1 -23661.99,E2 -23661.99} C_VEL
LIN {X 0,Y 173.232,Z 686.298,A -85,B 0,C 180,E1 -23663.598,E2 -23663.598} C_VEL
LIN {X 0,Y 174.907,Z 672.825,A -85,B 0,C 180,E1 -23664.889,E2 -23664.889} C_VEL
LIN {X 0,Y 176.113,Z 660.59,A -85,B 0,C 180,E1 -23665.628,E2 -23665.628} C_VEL
LIN {X 0,Y 179.207,Z 611.63,A -85,B 0,C 180,E1 -23667.706,E2 -23667.706} C_VEL
LIN {X 0,Y 173.065,Z 594.633,A -85,B 0,C 180,E1 -23669.773,E2 -23669.773} C_VEL
LIN {X 0,Y 163.863,Z 575.789,A -85,B 0,C 180,E1 -23672.781,E2 -23672.781} C_VEL
LIN {X 0,Y 159.411,Z 568.526,A -85,B 0,C 180,E1 -23674.271,E2 -23674.271} C_VEL
LIN {X 0,Y 157.979,Z 565.957,A -85,B 0,C 180,E1 -23674.789,E2 -23674.789} C_VEL
LIN {X 0,Y 157.738,Z 564.824,A -85,B 0,C 180,E1 -23674.956,E2 -23674.956} C_VEL
LIN {X 0,Y 157.812,Z 564.826,A -85,B 0,C 180,E1 -23677.681,E2 -23677.681} C_VEL
LIN {X 0,Y 157.675,Z 564.831,A -85,B 0,C 180,E1 -23681.312,E2 -23681.312} C_VEL
LIN {X 0,Y 157.479,Z 564.865,A -85,B 0,C 180,E1 -23685.535,E2 -23685.535} C_VEL
LIN {X 0,Y 157.371,Z 564.855,A -85,B 0,C 180,E1 -23690.936,E2 -23690.936} C_VEL
LIN {X 0,Y 157.316,Z 564.886,A -85,B 0,C 180,E1 -23696.688,E2 -23696.688} C_VEL
LIN {X 0,Y 157.277,Z 564.883,A -85,B 0,C 180,E1 -23702.431,E2 -23702.431} C_VEL
LIN {X 0,Y 157.271,Z 564.896,A -85,B 0,C 180,E1 -23706.453,E2 -23706.453} C_VEL
LIN {X 0,Y 157.214,Z 564.892,A -85,B 0,C 180,E1 -23712.114,E2 -23712.114} C_VEL
LIN {X 0,Y 157.215,Z 564.895,A -85,B 0,C 180,E1 -23717.893,E2 -23717.893} C_VEL
LIN {X 0,Y 157.273,Z 564.889,A -85,B 0,C 180,E1 -23723.554,E2 -23723.554} C_VEL
LIN {X 0,Y 157.3,Z 564.885,A -85,B 0,C 180,E1 -23728.099,E2 -23728.099} C_VEL
LIN {X 0,Y 157.322,Z 564.876,A -85,B 0,C 180,E1 -23733.468,E2 -23733.468} C_VEL
LIN {X 0,Y 157.398,Z 564.871,A -85,B 0,C 180,E1 -23739.673,E2 -23739.673} C_VEL
LIN {X 0,Y 157.442,Z 564.86,A -85,B 0,C 180,E1 -23744.466,E2 -23744.466} C_VEL
LIN {X 0,Y 157.698,Z 564.838,A -85,B 0,C 180,E1 -23749.733,E2 -23749.733} C_VEL
LIN {X 0,Y 157.776,Z 564.816,A -85,B 0,C 180,E1 -23752.322,E2 -23752.322} C_VEL
LIN {X 0,Y 158.267,Z 564.769,A -85,B 0,C 180,E1 -23760.001,E2 -23760.001} C_VEL
LIN {X 0,Y 157.83,Z 564.824,A -85,B 0,C 180,E1 -23767.678,E2 -23767.678} C_VEL
LIN {X 0,Y 157.689,Z 564.836,A -85,B 0,C 180,E1 -23771.314,E2 -23771.314} C_VEL
LIN {X 0,Y 157.466,Z 564.869,A -85,B 0,C 180,E1 -23775.534,E2 -23775.534} C_VEL
LIN {X 0,Y 157.378,Z 564.864,A -85,B 0,C 180,E1 -23780.933,E2 -23780.933} C_VEL
LIN {X 0,Y 157.319,Z 564.869,A -85,B 0,C 180,E1 -23786.68,E2 -23786.68} C_VEL
LIN {X 0,Y 157.285,Z 564.889,A -85,B 0,C 180,E1 -23792.427,E2 -23792.427} C_VEL
LIN {X 0,Y 157.277,Z 564.893,A -85,B 0,C 180,E1 -23796.448,E2 -23796.448} C_VEL
LIN {X 0,Y 157.202,Z 564.902,A -85,B 0,C 180,E1 -23802.115,E2 -23802.115} C_VEL
LIN {X 0,Y 157.247,Z 564.92,A -85,B 0,C 180,E1 -23804.127,E2 -23804.127} C_VEL
LIN {X 0,Y 157.35,Z 565.557,A -85,B 0,C 180,E1 -23804.562,E2 -23804.562} C_VEL
LIN {X 0,Y 159.21,Z 569.422,A -85,B 0,C 180,E1 -23805.271,E2 -23805.271} C_VEL
LIN {X 0,Y 166.506,Z 585.06,A -85,B 0,C 180,E1 -23807.883,E2 -23807.883} C_VEL
LIN {X 0,Y 172.549,Z 600.27,A -85,B 0,C 180,E1 -23809.973,E2 -23809.973} C_VEL
LIN {X 0,Y 177.322,Z 614.138,A -85,B 0,C 180,E1 -23811.626,E2 -23811.626} C_VEL
LIN {X 0,Y 178.603,Z 626.134,A -85,B 0,C 180,E1 -23812.487,E2 -23812.487} C_VEL
LIN {X 0,Y 175.571,Z 674.465,A -85,B 0,C 180,E1 -23814.604,E2 -23814.604} C_VEL
LIN {X 0,Y 174.098,Z 686.885,A -85,B 0,C 180,E1 -23815.496,E2 -23815.496} C_VEL
LIN {X 0,Y 172.193,Z 698.766,A -85,B 0,C 180,E1 -23816.736,E2 -23816.736} C_VEL
LIN {X 0,Y 170.214,Z 709.343,A -85,B 0,C 180,E1 -23818.231,E2 -23818.231} C_VEL
LIN {X 0,Y 167.736,Z 720.047,A -85,B 0,C 180,E1 -23820.158,E2 -23820.158} C_VEL
LIN {X 0,Y 164.942,Z 731.055,A -85,B 0,C 180,E1 -23822.735,E2 -23822.735} C_VEL
LIN {X 0,Y 162.331,Z 740.493,A -85,B 0,C 180,E1 -23825.544,E2 -23825.544} C_VEL
LIN {X 0,Y 160.451,Z 747.545,A -85,B 0,C 180,E1 -23828.138,E2 -23828.138} C_VEL
LIN {X 0,Y 158.178,Z 755.758,A -85,B 0,C 180,E1 -23831.876,E2 -23831.876} C_VEL
LIN {X 0,Y 156.47,Z 762.168,A -85,B 0,C 180,E1 -23835.597,E2 -23835.597} C_VEL
LIN {X 0,Y 155.267,Z 764.907,A -85,B 0,C 180,E1 -23837.467,E2 -23837.467} C_VEL
LIN {X 0,Y 151.727,Z 768.6,A -85,B 0,C 180,E1 -23840.637,E2 -23840.637} C_VEL
LIN {X 0,Y 148.958,Z 771.068,A -85,B 0,C 180,E1 -23843.351,E2 -23843.351} C_VEL
LIN {X 0,Y 147.79,Z 772.711,A -85,B 0,C 180,E1 -23845.523,E2 -23845.523} C_VEL
LIN {X 0,Y 147.691,Z 773.152,A -85,B 0,C 180,E1 -23846.266,E2 -23846.266} C_VEL
LIN {X 0,Y 147.78,Z 775.281,A -85,B 0,C 180,E1 -23849.996,E2 -23849.996} C_VEL
LIN {X 0,Y 147.64,Z 776.251,A -85,B 0,C 180,E1 -23852.725,E2 -23852.725} C_VEL
LIN {X 0,Y 147.692,Z 776.831,A -85,B 0,C 180,E1 -23855.457,E2 -23855.457} C_VEL
LIN {X 0,Y 147.94,Z 777.026,A -85,B 0,C 180,E1 -23858.19,E2 -23858.19} C_VEL
LIN {X 0,Y 148.431,Z 776.831,A -85,B 0,C 180,E1 -23860.913,E2 -23860.913} C_VEL
LIN {X 0,Y 150.319,Z 775.239,A -85,B 0,C 180,E1 -23866.287,E2 -23866.287} C_VEL
LIN {X 0,Y 151.73,Z 773.876,A -85,B 0,C 180,E1 -23868.915,E2 -23868.915} C_VEL
LIN {X 0,Y 154.628,Z 771.047,A -85,B 0,C 180,E1 -23872.722,E2 -23872.722} C_VEL
LIN {X 0,Y 158.079,Z 767.241,A -85,B 0,C 180,E1 -23876.393,E2 -23876.393} C_VEL
LIN {X 0,Y 162.187,Z 762.329,A -85,B 0,C 180,E1 -23879.925,E2 -23879.925} C_VEL
LIN {X 0,Y 166.848,Z 756.335,A -85,B 0,C 180,E1 -23883.197,E2 -23883.197} C_VEL
LIN {X 0,Y 172.139,Z 748.883,A -85,B 0,C 180,E1 -23886.294,E2 -23886.294} C_VEL
LIN {X 0,Y 177.002,Z 741.33,A -85,B 0,C 180,E1 -23888.705,E2 -23888.705} C_VEL
LIN {X 0,Y 182.63,Z 731.244,A -85,B 0,C 180,E1 -23891.219,E2 -23891.219} C_VEL
LIN {X 0,Y 188.235,Z 719.826,A -85,B 0,C 180,E1 -23893.314,E2 -23893.314} C_VEL
LIN {X 0,Y 192.878,Z 708.421,A -85,B 0,C 180,E1 -23894.904,E2 -23894.904} C_VEL
LIN {X 0,Y 197.127,Z 695.436,A -85,B 0,C 180,E1 -23896.212,E2 -23896.212} C_VEL
LIN {X 0,Y 200.282,Z 682.95,A -85,B 0,C 180,E1 -23897.093,E2 -23897.093} C_VEL
LIN {X 0,Y 202.567,Z 668.886,A -85,B 0,C 180,E1 -23897.781,E2 -23897.781} C_VEL
LIN {X 0,Y 205.371,Z 641.82,A -85,B 0,C 180,E1 -23898.744,E2 -23898.744} C_VEL
LIN {X 0,Y 202.899,Z 634.639,A -85,B 0,C 180,E1 -23900.795,E2 -23900.795} C_VEL
LIN {X 0,Y 199.889,Z 627.47,A -85,B 0,C 180,E1 -23903.507,E2 -23903.507} C_VEL
LIN {X 0,Y 198.09,Z 623.426,A -85,B 0,C 180,E1 -23905.412,E2 -23905.412} C_VEL
LIN {X 0,Y 196.589,Z 620.301,A -85,B 0,C 180,E1 -23907.158,E2 -23907.158} C_VEL
LIN {X 0,Y 194.686,Z 616.235,A -85,B 0,C 180,E1 -23909.908,E2 -23909.908} C_VEL
LIN {X 0,Y 192.092,Z 610.911,A -85,B 0,C 180,E1 -23915.827,E2 -23915.827} C_VEL
LIN {X 0,Y 191.522,Z 609.825,A -85,B 0,C 180,E1 -23920.714,E2 -23920.714} C_VEL
LIN {X 0,Y 192.138,Z 610.093,A -85,B 0,C 180,E1 -23924.458,E2 -23924.458} C_VEL
LIN {X 0,Y 194.599,Z 613.587,A -85,B 0,C 180,E1 -23929.977,E2 -23929.977} C_VEL
LIN {X 0,Y 196.67,Z 617.095,A -85,B 0,C 180,E1 -23932.959,E2 -23932.959} C_VEL
LIN {X 0,Y 197.794,Z 618.471,A -85,B 0,C 180,E1 -23934.175,E2 -23934.175} C_VEL
LIN {X 0,Y 199.93,Z 623.013,A -85,B 0,C 180,E1 -23936.499,E2 -23936.499} C_VEL
LIN {X 0,Y 202.631,Z 628.363,A -85,B 0,C 180,E1 -23938.909,E2 -23938.909} C_VEL
LIN {X 0,Y 205.805,Z 636.262,A -85,B 0,C 180,E1 -23941.499,E2 -23941.499} C_VEL
LIN {X 0,Y 202.36,Z 668.244,A -85,B 0,C 180,E1 -23942.68,E2 -23942.68} C_VEL
LIN {X 0,Y 199.771,Z 681.909,A -85,B 0,C 180,E1 -23943.473,E2 -23943.473} C_VEL
LIN {X 0,Y 196.414,Z 694.595,A -85,B 0,C 180,E1 -23944.597,E2 -23944.597} C_VEL
LIN {X 0,Y 192.027,Z 707.334,A -85,B 0,C 180,E1 -23946.154,E2 -23946.154} C_VEL
LIN {X 0,Y 187.16,Z 718.581,A -85,B 0,C 180,E1 -23947.977,E2 -23947.977} C_VEL
LIN {X 0,Y 182.045,Z 728.656,A -85,B 0,C 180,E1 -23950.145,E2 -23950.145} C_VEL
LIN {X 0,Y 176.518,Z 738.03,A -85,B 0,C 180,E1 -23952.742,E2 -23952.742} C_VEL
LIN {X 0,Y 171.378,Z 745.637,A -85,B 0,C 180,E1 -23955.502,E2 -23955.502} C_VEL
LIN {X 0,Y 166.691,Z 751.888,A -85,B 0,C 180,E1 -23958.455,E2 -23958.455} C_VEL
LIN {X 0,Y 161.439,Z 758.065,A -85,B 0,C 180,E1 -23962.345,E2 -23962.345} C_VEL
LIN {X 0,Y 156.854,Z 762.9,A -85,B 0,C 180,E1 -23966.618,E2 -23966.618} C_VEL
LIN {X 0,Y 153.94,Z 765.639,A -85,B 0,C 180,E1 -23970.144,E2 -23970.144} C_VEL
LIN {X 0,Y 151.492,Z 767.577,A -85,B 0,C 180,E1 -23973.826,E2 -23973.826} C_VEL
LIN {X 0,Y 149.661,Z 768.709,A -85,B 0,C 180,E1 -23977.622,E2 -23977.622} C_VEL
LIN {X 0,Y 148.314,Z 769.045,A -85,B 0,C 180,E1 -23981.558,E2 -23981.558} C_VEL
LIN {X 0,Y 147.491,Z 768.5,A -85,B 0,C 180,E1 -23985.621,E2 -23985.621} C_VEL
LIN {X 0,Y 147.157,Z 767.013,A -85,B 0,C 180,E1 -23989.828,E2 -23989.828} C_VEL
LIN {X 0,Y 147.484,Z 763.745,A -85,B 0,C 180,E1 -23995.127,E2 -23995.127} C_VEL
LIN {X 0,Y 148.155,Z 760.656,A -85,B 0,C 180,E1 -23998.632,E2 -23998.632} C_VEL
LIN {X 0,Y 149.444,Z 755.127,A -85,B 0,C 180,E1 -24003.316,E2 -24003.316} C_VEL
LIN {X 0,Y 151.212,Z 748.703,A -85,B 0,C 180,E1 -24007.459,E2 -24007.459} C_VEL
LIN {X 0,Y 153.412,Z 741.105,A -85,B 0,C 180,E1 -24011.3,E2 -24011.3} C_VEL
LIN {X 0,Y 155.925,Z 732.694,A -85,B 0,C 180,E1 -24014.649,E2 -24014.649} C_VEL
LIN {X 0,Y 158.387,Z 723.861,A -85,B 0,C 180,E1 -24017.466,E2 -24017.466} C_VEL
LIN {X 0,Y 161.31,Z 712.891,A -85,B 0,C 180,E1 -24020.221,E2 -24020.221} C_VEL
LIN {X 0,Y 163.886,Z 701.544,A -85,B 0,C 180,E1 -24022.447,E2 -24022.447} C_VEL
LIN {X 0,Y 166.25,Z 689.332,A -85,B 0,C 180,E1 -24024.241,E2 -24024.241} C_VEL
LIN {X 0,Y 168.212,Z 676.289,A -85,B 0,C 180,E1 -24025.639,E2 -24025.639} C_VEL
LIN {X 0,Y 169.599,Z 663.119,A -85,B 0,C 180,E1 -24026.566,E2 -24026.566} C_VEL
LIN {X 0,Y 172.853,Z 613.168,A -85,B 0,C 180,E1 -24028.783,E2 -24028.783} C_VEL
LIN {X 0,Y 167.4,Z 597.97,A -85,B 0,C 180,E1 -24030.7,E2 -24030.7} C_VEL
LIN {X 0,Y 158.852,Z 580.139,A -85,B 0,C 180,E1 -24033.674,E2 -24033.674} C_VEL
LIN {X 0,Y 152.193,Z 569.284,A -85,B 0,C 180,E1 -24036.056,E2 -24036.056} C_VEL
LIN {X 0,Y 150.84,Z 566.516,A -85,B 0,C 180,E1 -24036.609,E2 -24036.609} C_VEL
LIN {X 0,Y 150.698,Z 565.704,A -85,B 0,C 180,E1 -24036.783,E2 -24036.783} C_VEL
LIN {X 0,Y 150.61,Z 565.708,A -85,B 0,C 180,E1 -24041.504,E2 -24041.504} C_VEL
LIN {X 0,Y 150.384,Z 565.752,A -85,B 0,C 180,E1 -24046.288,E2 -24046.288} C_VEL
LIN {X 0,Y 150.351,Z 565.729,A -85,B 0,C 180,E1 -24050.796,E2 -24050.796} C_VEL
LIN {X 0,Y 150.246,Z 565.769,A -85,B 0,C 180,E1 -24057.286,E2 -24057.286} C_VEL
LIN {X 0,Y 150.217,Z 565.762,A -85,B 0,C 180,E1 -24062.636,E2 -24062.636} C_VEL
LIN {X 0,Y 150.176,Z 565.779,A -85,B 0,C 180,E1 -24067.477,E2 -24067.477} C_VEL
LIN {X 0,Y 150.153,Z 565.768,A -85,B 0,C 180,E1 -24071.508,E2 -24071.508} C_VEL
LIN {X 0,Y 150.13,Z 565.786,A -85,B 0,C 180,E1 -24075.399,E2 -24075.399} C_VEL
LIN {X 0,Y 150.155,Z 565.766,A -85,B 0,C 180,E1 -24079.062,E2 -24079.062} C_VEL
LIN {X 0,Y 150.184,Z 565.769,A -85,B 0,C 180,E1 -24082.711,E2 -24082.711} C_VEL
LIN {X 0,Y 150.221,Z 565.77,A -85,B 0,C 180,E1 -24087.371,E2 -24087.371} C_VEL
LIN {X 0,Y 150.248,Z 565.753,A -85,B 0,C 180,E1 -24092.723,E2 -24092.723} C_VEL
LIN {X 0,Y 150.356,Z 565.751,A -85,B 0,C 180,E1 -24099.213,E2 -24099.213} C_VEL
LIN {X 0,Y 150.351,Z 565.736,A -85,B 0,C 180,E1 -24103.714,E2 -24103.714} C_VEL
LIN {X 0,Y 150.62,Z 565.722,A -85,B 0,C 180,E1 -24109.245,E2 -24109.245} C_VEL
LIN {X 0,Y 150.714,Z 565.697,A -85,B 0,C 180,E1 -24111.96,E2 -24111.96} C_VEL
LIN {X 0,Y 151.227,Z 565.646,A -85,B 0,C 180,E1 -24120.001,E2 -24120.001} C_VEL
LIN {X 0,Y 150.766,Z 565.706,A -85,B 0,C 180,E1 -24128.04,E2 -24128.04} C_VEL
LIN {X 0,Y 150.624,Z 565.714,A -85,B 0,C 180,E1 -24131.507,E2 -24131.507} C_VEL
LIN {X 0,Y 150.374,Z 565.756,A -85,B 0,C 180,E1 -24136.287,E2 -24136.287} C_VEL
LIN {X 0,Y 150.36,Z 565.739,A -85,B 0,C 180,E1 -24140.791,E2 -24140.791} C_VEL
LIN {X 0,Y 150.251,Z 565.755,A -85,B 0,C 180,E1 -24147.279,E2 -24147.279} C_VEL
LIN {X 0,Y 150.224,Z 565.769,A -85,B 0,C 180,E1 -24152.631,E2 -24152.631} C_VEL
LIN {X 0,Y 150.182,Z 565.78,A -85,B 0,C 180,E1 -24157.472,E2 -24157.472} C_VEL
LIN {X 0,Y 150.199,Z 565.894,A -85,B 0,C 180,E1 -24162.691,E2 -24162.691} C_VEL
LIN {X 0,Y 151.219,Z 568.617,A -85,B 0,C 180,E1 -24163.156,E2 -24163.156} C_VEL
LIN {X 0,Y 152.816,Z 571.149,A -85,B 0,C 180,E1 -24163.751,E2 -24163.751} C_VEL
LIN {X 0,Y 157.226,Z 580.167,A -85,B 0,C 180,E1 -24165.468,E2 -24165.468} C_VEL
LIN {X 0,Y 163.576,Z 594.734,A -85,B 0,C 180,E1 -24167.831,E2 -24167.831} C_VEL
LIN {X 0,Y 171.019,Z 615.258,A -85,B 0,C 180,E1 -24170.519,E2 -24170.519} C_VEL
LIN {X 0,Y 172.338,Z 626.869,A -85,B 0,C 180,E1 -24171.413,E2 -24171.413} C_VEL
LIN {X 0,Y 169.169,Z 674.932,A -85,B 0,C 180,E1 -24173.593,E2 -24173.593} C_VEL
LIN {X 0,Y 167.523,Z 687.953,A -85,B 0,C 180,E1 -24174.583,E2 -24174.583} C_VEL
LIN {X 0,Y 165.472,Z 700.063,A -85,B 0,C 180,E1 -24175.933,E2 -24175.933} C_VEL
LIN {X 0,Y 163.03,Z 711.903,A -85,B 0,C 180,E1 -24177.756,E2 -24177.756} C_VEL
LIN {X 0,Y 160.243,Z 723.346,A -85,B 0,C 180,E1 -24180.07,E2 -24180.07} C_VEL
LIN {X 0,Y 157.475,Z 733.727,A -85,B 0,C 180,E1 -24182.773,E2 -24182.773} C_VEL
LIN {X 0,Y 154.69,Z 743.023,A -85,B 0,C 180,E1 -24185.861,E2 -24185.861} C_VEL
LIN {X 0,Y 152.489,Z 750.716,A -85,B 0,C 180,E1 -24189.069,E2 -24189.069} C_VEL
LIN {X 0,Y 150.374,Z 758.232,A -85,B 0,C 180,E1 -24193.012,E2 -24193.012} C_VEL
LIN {X 0,Y 149.1,Z 763.318,A -85,B 0,C 180,E1 -24196.364,E2 -24196.364} C_VEL
LIN {X 0,Y 148.206,Z 768.227,A -85,B 0,C 180,E1 -24200.442,E2 -24200.442} C_VEL
LIN {X 0,Y 147.783,Z 771.951,A -85,B 0,C 180,E1 -24204.538,E2 -24204.538} C_VEL
LIN {X 0,Y 147.691,Z 773.152,A -85,B 0,C 180,E1 -24206.266,E2 -24206.266} C_VEL
LIN {X 0,Y 146.968,Z 774.502,A -85,B 0,C 180,E1 -24208.48,E2 -24208.48} C_VEL
LIN {X 0,Y 145.327,Z 775.447,A -85,B 0,C 180,E1 -24210.688,E2 -24210.688} C_VEL
LIN {X 0,Y 141.671,Z 776.515,A -85,B 0,C 180,E1 -24215.253,E2 -24215.253} C_VEL
LIN {X 0,Y 140.851,Z 776.76,A -85,B 0,C 180,E1 -24217.664,E2 -24217.664} C_VEL
LIN {X 0,Y 140.884,Z 776.775,A -85,B 0,C 180,E1 -24218.477,E2 -24218.477} C_VEL
LIN {X 0,Y 141.443,Z 776.664,A -85,B 0,C 180,E1 -24221.46,E2 -24221.46} C_VEL
LIN {X 0,Y 142.315,Z 776.165,A -85,B 0,C 180,E1 -24224.291,E2 -24224.291} C_VEL
LIN {X 0,Y 145.024,Z 773.951,A -85,B 0,C 180,E1 -24229.825,E2 -24229.825} C_VEL
LIN {X 0,Y 149.309,Z 770.175,A -85,B 0,C 180,E1 -24235.06,E2 -24235.06} C_VEL
LIN {X 0,Y 153.106,Z 766.192,A -85,B 0,C 180,E1 -24238.81,E2 -24238.81} C_VEL
LIN {X 0,Y 157.569,Z 761.136,A -85,B 0,C 180,E1 -24242.355,E2 -24242.355} C_VEL
LIN {X 0,Y 162.805,Z 754.834,A -85,B 0,C 180,E1 -24245.641,E2 -24245.641} C_VEL
LIN {X 0,Y 168.506,Z 747.05,A -85,B 0,C 180,E1 -24248.723,E2 -24248.723} C_VEL
LIN {X 0,Y 174.761,Z 737.492,A -85,B 0,C 180,E1 -24251.566,E2 -24251.566} C_VEL
LIN {X 0,Y 180.305,Z 727.71,A -85,B 0,C 180,E1 -24253.773,E2 -24253.773} C_VEL
LIN {X 0,Y 185.608,Z 716.772,A -85,B 0,C 180,E1 -24255.614,E2 -24255.614} C_VEL
LIN {X 0,Y 190.526,Z 704.555,A -85,B 0,C 180,E1 -24257.145,E2 -24257.145} C_VEL
LIN {X 0,Y 194.314,Z 692.687,A -85,B 0,C 180,E1 -24258.237,E2 -24258.237} C_VEL
LIN {X 0,Y 197.589,Z 679.058,A -85,B 0,C 180,E1 -24259.08,E2 -24259.08} C_VEL
LIN {X 0,Y 199.597,Z 665.729,A -85,B 0,C 180,E1 -24259.675,E2 -24259.675} C_VEL
LIN {X 0,Y 201.807,Z 644.687,A -85,B 0,C 180,E1 -24260.446,E2 -24260.446} C_VEL
LIN {X 0,Y 199.547,Z 638.017,A -85,B 0,C 180,E1 -24262.564,E2 -24262.564} C_VEL
LIN {X 0,Y 196.587,Z 630.597,A -85,B 0,C 180,E1 -24265.711,E2 -24265.711} C_VEL
LIN {X 0,Y 194.799,Z 626.657,A -85,B 0,C 180,E1 -24267.927,E2 -24267.927} C_VEL
LIN {X 0,Y 193.081,Z 622.7,A -85,B 0,C 180,E1 -24270.671,E2 -24270.671} C_VEL
LIN {X 0,Y 190.932,Z 617.848,A -85,B 0,C 180,E1 -24276.114,E2 -24276.114} C_VEL
LIN {X 0,Y 190.445,Z 616.865,A -85,B 0,C 180,E1 -24280.601,E2 -24280.601} C_VEL
LIN {X 0,Y 191.032,Z 617.185,A -85,B 0,C 180,E1 -24284.366,E2 -24284.366} C_VEL
LIN {X 0,Y 193.133,Z 620.323,A -85,B 0,C 180,E1 -24289.424,E2 -24289.424} C_VEL
LIN {X 0,Y 195.168,Z 623.842,A -85,B 0,C 180,E1 -24292.499,E2 -24292.499} C_VEL
LIN {X 0,Y 196.091,Z 625.151,A -85,B 0,C 180,E1 -24293.605,E2 -24293.605} C_VEL
LIN {X 0,Y 199.183,Z 631.89,A -85,B 0,C 180,E1 -24297.018,E2 -24297.018} C_VEL
LIN {X 0,Y 201.286,Z 637.02,A -85,B 0,C 180,E1 -24298.963,E2 -24298.963} C_VEL
LIN {X 0,Y 202.281,Z 639.867,A -85,B 0,C 180,E1 -24299.863,E2 -24299.863} C_VEL
LIN {X 0,Y 198.97,Z 668.552,A -85,B 0,C 180,E1 -24300.904,E2 -24300.904} C_VEL
LIN {X 0,Y 196.313,Z 682.002,A -85,B 0,C 180,E1 -24301.678,E2 -24301.678} C_VEL
LIN {X 0,Y 192.953,Z 694.304,A -85,B 0,C 180,E1 -24302.745,E2 -24302.745} C_VEL
LIN {X 0,Y 188.362,Z 707.174,A -85,B 0,C 180,E1 -24304.278,E2 -24304.278} C_VEL
LIN {X 0,Y 183.702,Z 717.708,A -85,B 0,C 180,E1 -24305.937,E2 -24305.937} C_VEL
LIN {X 0,Y 178.303,Z 727.945,A -85,B 0,C 180,E1 -24308.065,E2 -24308.065} C_VEL
LIN {X 0,Y 172.478,Z 737.416,A -85,B 0,C 180,E1 -24310.65,E2 -24310.65} C_VEL
LIN {X 0,Y 166.392,Z 745.958,A -85,B 0,C 180,E1 -24313.737,E2 -24313.737} C_VEL
LIN {X 0,Y 160.332,Z 753.452,A -85,B 0,C 180,E1 -24317.439,E2 -24317.439} C_VEL
LIN {X 0,Y 155.094,Z 759.112,A -85,B 0,C 180,E1 -24321.253,E2 -24321.253} C_VEL
LIN {X 0,Y 151.189,Z 762.852,A -85,B 0,C 180,E1 -24324.73,E2 -24324.73} C_VEL
LIN {X 0,Y 147.971,Z 765.654,A -85,B 0,C 180,E1 -24328.355,E2 -24328.355} C_VEL
LIN {X 0,Y 144.152,Z 768.349,A -85,B 0,C 180,E1 -24334.03,E2 -24334.03} C_VEL
LIN {X 0,Y 142.402,Z 769.138,A -85,B 0,C 180,E1 -24337.854,E2 -24337.854} C_VEL
LIN {X 0,Y 141.141,Z 769.185,A -85,B 0,C 180,E1 -24341.683,E2 -24341.683} C_VEL
LIN {X 0,Y 140.403,Z 768.554,A -85,B 0,C 180,E1 -24345.517,E2 -24345.517} C_VEL
LIN {X 0,Y 140.055,Z 766.301,A -85,B 0,C 180,E1 -24351.158,E2 -24351.158} C_VEL
LIN {X 0,Y 140.617,Z 762.573,A -85,B 0,C 180,E1 -24356.654,E2 -24356.654} C_VEL
LIN {X 0,Y 141.384,Z 759.192,A -85,B 0,C 180,E1 -24360.198,E2 -24360.198} C_VEL
LIN {X 0,Y 142.706,Z 754.002,A -85,B 0,C 180,E1 -24364.479,E2 -24364.479} C_VEL
LIN {X 0,Y 144.61,Z 747.514,A -85,B 0,C 180,E1 -24368.641,E2 -24368.641} C_VEL
LIN {X 0,Y 147.131,Z 739.133,A -85,B 0,C 180,E1 -24372.806,E2 -24372.806} C_VEL
LIN {X 0,Y 149.983,Z 729.738,A -85,B 0,C 180,E1 -24376.454,E2 -24376.454} C_VEL
LIN {X 0,Y 152.777,Z 720.03,A -85,B 0,C 180,E1 -24379.401,E2 -24379.401} C_VEL
LIN {X 0,Y 155.943,Z 707.939,A -85,B 0,C 180,E1 -24382.233,E2 -24382.233} C_VEL
LIN {X 0,Y 158.656,Z 695.463,A -85,B 0,C 180,E1 -24384.443,E2 -24384.443} C_VEL
LIN {X 0,Y 160.974,Z 682.609,A -85,B 0,C 180,E1 -24386.098,E2 -24386.098} C_VEL
LIN {X 0,Y 162.665,Z 669.494,A -85,B 0,C 180,E1 -24387.283,E2 -24387.283} C_VEL
LIN {X 0,Y 164.072,Z 652.565,A -85,B 0,C 180,E1 -24388.178,E2 -24388.178} C_VEL
LIN {X 0,Y 166.622,Z 614.743,A -85,B 0,C 180,E1 -24389.879,E2 -24389.879} C_VEL
LIN {X 0,Y 161.802,Z 601.344,A -85,B 0,C 180,E1 -24391.686,E2 -24391.686} C_VEL
LIN {X 0,Y 153.79,Z 584.439,A -85,B 0,C 180,E1 -24394.631,E2 -24394.631} C_VEL
LIN {X 0,Y 145.073,Z 569.95,A -85,B 0,C 180,E1 -24397.995,E2 -24397.995} C_VEL
LIN {X 0,Y 143.804,Z 567.289,A -85,B 0,C 180,E1 -24398.568,E2 -24398.568} C_VEL
LIN {X 0,Y 143.642,Z 566.596,A -85,B 0,C 180,E1 -24398.799,E2 -24398.799} C_VEL
LIN {X 0,Y 143.547,Z 566.586,A -85,B 0,C 180,E1 -24401.717,E2 -24401.717} C_VEL
LIN {X 0,Y 143.317,Z 566.634,A -85,B 0,C 180,E1 -24407.115,E2 -24407.115} C_VEL
LIN {X 0,Y 143.277,Z 566.605,A -85,B 0,C 180,E1 -24411.258,E2 -24411.258} C_VEL
LIN {X 0,Y 143.192,Z 566.651,A -85,B 0,C 180,E1 -24417.941,E2 -24417.941} C_VEL
LIN {X 0,Y 143.145,Z 566.646,A -85,B 0,C 180,E1 -24423.424,E2 -24423.424} C_VEL
LIN {X 0,Y 143.064,Z 566.652,A -85,B 0,C 180,E1 -24429.694,E2 -24429.694} C_VEL
LIN {X 0,Y 143.06,Z 566.661,A -85,B 0,C 180,E1 -24433.459,E2 -24433.459} C_VEL
LIN {X 0,Y 143.07,Z 566.658,A -85,B 0,C 180,E1 -24437.469,E2 -24437.469} C_VEL
LIN {X 0,Y 143.082,Z 566.645,A -85,B 0,C 180,E1 -24441.81,E2 -24441.81} C_VEL
LIN {X 0,Y 143.188,Z 566.646,A -85,B 0,C 180,E1 -24447.325,E2 -24447.325} C_VEL
LIN {X 0,Y 143.195,Z 566.627,A -85,B 0,C 180,E1 -24452.068,E2 -24452.068} C_VEL
LIN {X 0,Y 143.282,Z 566.634,A -85,B 0,C 180,E1 -24458.751,E2 -24458.751} C_VEL
LIN {X 0,Y 143.289,Z 566.612,A -85,B 0,C 180,E1 -24462.887,E2 -24462.887} C_VEL
LIN {X 0,Y 143.546,Z 566.603,A -85,B 0,C 180,E1 -24468.708,E2 -24468.708} C_VEL
LIN {X 0,Y 143.635,Z 566.58,A -85,B 0,C 180,E1 -24471.561,E2 -24471.561} C_VEL
LIN {X 0,Y 144.186,Z 566.523,A -85,B 0,C 180,E1 -24480.001,E2 -24480.001} C_VEL
LIN {X 0,Y 143.685,Z 566.588,A -85,B 0,C 180,E1 -24488.439,E2 -24488.439} C_VEL
LIN {X 0,Y 143.558,Z 566.592,A -85,B 0,C 180,E1 -24491.713,E2 -24491.713} C_VEL
LIN {X 0,Y 143.312,Z 566.635,A -85,B 0,C 180,E1 -24497.113,E2 -24497.113} C_VEL
LIN {X 0,Y 143.285,Z 566.613,A -85,B 0,C 180,E1 -24501.252,E2 -24501.252} C_VEL
LIN {X 0,Y 143.198,Z 566.64,A -85,B 0,C 180,E1 -24507.935,E2 -24507.935} C_VEL
LIN {X 0,Y 143.153,Z 566.653,A -85,B 0,C 180,E1 -24513.419,E2 -24513.419} C_VEL
LIN {X 0,Y 143.065,Z 566.663,A -85,B 0,C 180,E1 -24519.691,E2 -24519.691} C_VEL
LIN {X 0,Y 143.107,Z 566.66,A -85,B 0,C 180,E1 -24520.664,E2 -24520.664} C_VEL
LIN {X 0,Y 144.236,Z 569.716,A -85,B 0,C 180,E1 -24521.269,E2 -24521.269} C_VEL
LIN {X 0,Y 145.661,Z 571.731,A -85,B 0,C 180,E1 -24521.83,E2 -24521.83} C_VEL
LIN {X 0,Y 149.566,Z 578.789,A -85,B 0,C 180,E1 -24523.412,E2 -24523.412} C_VEL
LIN {X 0,Y 155.883,Z 592.794,A -85,B 0,C 180,E1 -24525.948,E2 -24525.948} C_VEL
LIN {X 0,Y 161.986,Z 608.824,A -85,B 0,C 180,E1 -24528.338,E2 -24528.338} C_VEL
LIN {X 0,Y 165.123,Z 618.019,A -85,B 0,C 180,E1 -24529.537,E2 -24529.537} C_VEL
LIN {X 0,Y 166.026,Z 627.879,A -85,B 0,C 180,E1 -24530.289,E2 -24530.289} C_VEL
LIN {X 0,Y 162.851,Z 674.524,A -85,B 0,C 180,E1 -24532.478,E2 -24532.478} C_VEL
LIN {X 0,Y 161.117,Z 687.911,A -85,B 0,C 180,E1 -24533.531,E2 -24533.531} C_VEL
LIN {X 0,Y 159.198,Z 698.872,A -85,B 0,C 180,E1 -24534.78,E2 -24534.78} C_VEL
LIN {X 0,Y 156.662,Z 710.997,A -85,B 0,C 180,E1 -24536.66,E2 -24536.66} C_VEL
LIN {X 0,Y 153.76,Z 722.566,A -85,B 0,C 180,E1 -24539.051,E2 -24539.051} C_VEL
LIN {X 0,Y 150.842,Z 733.045,A -85,B 0,C 180,E1 -24541.849,E2 -24541.849} C_VEL
LIN {X 0,Y 148.155,Z 741.595,A -85,B 0,C 180,E1 -24544.723,E2 -24544.723} C_VEL
LIN {X 0,Y 145.832,Z 749.514,A -85,B 0,C 180,E1 -24548.065,E2 -24548.065} C_VEL
LIN {X 0,Y 143.585,Z 757.211,A -85,B 0,C 180,E1 -24552.183,E2 -24552.183} C_VEL
LIN {X 0,Y 141.779,Z 764.292,A -85,B 0,C 180,E1 -24557.107,E2 -24557.107} C_VEL
LIN {X 0,Y 140.976,Z 768.937,A -85,B 0,C 180,E1 -24561.395,E2 -24561.395} C_VEL
LIN {X 0,Y 140.611,Z 772.753,A -85,B 0,C 180,E1 -24566.304,E2 -24566.304} C_VEL
LIN {X 0,Y 140.692,Z 774.846,A -85,B 0,C 180,E1 -24569.996,E2 -24569.996} C_VEL
LIN {X 0,Y 140.548,Z 775.896,A -85,B 0,C 180,E1 -24572.862,E2 -24572.862} C_VEL
LIN {X 0,Y 140.884,Z 776.775,A -85,B 0,C 180,E1 -24578.477,E2 -24578.477} C_VEL
LIN {X 0,Y 140.664,Z 776.834,A -85,B 0,C 180,E1 -24580.88,E2 -24580.88} C_VEL
LIN {X 0,Y 138.937,Z 776.288,A -85,B 0,C 180,E1 -24584.881,E2 -24584.881} C_VEL
LIN {X 0,Y 137.882,Z 774.949,A -85,B 0,C 180,E1 -24588.933,E2 -24588.933} C_VEL
LIN {X 0,Y 138.703,Z 773.766,A -85,B 0,C 180,E1 -24591.309,E2 -24591.309} C_VEL
LIN {X 0,Y 142.893,Z 770.425,A -85,B 0,C 180,E1 -24596.269,E2 -24596.269} C_VEL
LIN {X 0,Y 146.938,Z 766.591,A -85,B 0,C 180,E1 -24600.142,E2 -24600.142} C_VEL
LIN {X 0,Y 151.644,Z 761.7,A -85,B 0,C 180,E1 -24603.785,E2 -24603.785} C_VEL
LIN {X 0,Y 158.113,Z 754.505,A -85,B 0,C 180,E1 -24607.67,E2 -24607.67} C_VEL
LIN {X 0,Y 164.159,Z 746.734,A -85,B 0,C 180,E1 -24610.755,E2 -24610.755} C_VEL
LIN {X 0,Y 170.708,Z 737.155,A -85,B 0,C 180,E1 -24613.593,E2 -24613.593} C_VEL
LIN {X 0,Y 176.544,Z 727.324,A -85,B 0,C 180,E1 -24615.766,E2 -24615.766} C_VEL
LIN {X 0,Y 182.071,Z 716.394,A -85,B 0,C 180,E1 -24617.576,E2 -24617.576} C_VEL
LIN {X 0,Y 186.541,Z 705.892,A -85,B 0,C 180,E1 -24618.89,E2 -24618.89} C_VEL
LIN {X 0,Y 190.778,Z 693.519,A -85,B 0,C 180,E1 -24620.054,E2 -24620.054} C_VEL
LIN {X 0,Y 194.267,Z 680.002,A -85,B 0,C 180,E1 -24620.89,E2 -24620.89} C_VEL
LIN {X 0,Y 196.467,Z 666.422,A -85,B 0,C 180,E1 -24621.508,E2 -24621.508} C_VEL
LIN {X 0,Y 198.508,Z 647.863,A -85,B 0,C 180,E1 -24622.178,E2 -24622.178} C_VEL
LIN {X 0,Y 196.4,Z 641.671,A -85,B 0,C 180,E1 -24624.404,E2 -24624.404} C_VEL
LIN {X 0,Y 194.255,Z 635.898,A -85,B 0,C 180,E1 -24627.027,E2 -24627.027} C_VEL
LIN {X 0,Y 192.997,Z 632.857,A -85,B 0,C 180,E1 -24628.834,E2 -24628.834} C_VEL
LIN {X 0,Y 191.556,Z 629.275,A -85,B 0,C 180,E1 -24631.354,E2 -24631.354} C_VEL
LIN {X 0,Y 189.752,Z 624.728,A -85,B 0,C 180,E1 -24636.619,E2 -24636.619} C_VEL
LIN {X 0,Y 189.37,Z 623.906,A -85,B 0,C 180,E1 -24640.486,E2 -24640.486} C_VEL
LIN {X 0,Y 189.856,Z 623.996,A -85,B 0,C 180,E1 -24643.839,E2 -24643.839} C_VEL
LIN {X 0,Y 191.739,Z 627.172,A -85,B 0,C 180,E1 -24648.966,E2 -24648.966} C_VEL
LIN {X 0,Y 193.905,Z 630.872,A -85,B 0,C 180,E1 -24652.334,E2 -24652.334} C_VEL
LIN {X 0,Y 195.068,Z 633.309,A -85,B 0,C 180,E1 -24653.854,E2 -24653.854} C_VEL
LIN {X 0,Y 197.8,Z 639.783,A -85,B 0,C 180,E1 -24656.942,E2 -24656.942} C_VEL
LIN {X 0,Y 198.917,Z 643.027,A -85,B 0,C 180,E1 -24658.078,E2 -24658.078} C_VEL
LIN {X 0,Y 195.873,Z 668.877,A -85,B 0,C 180,E1 -24659.057,E2 -24659.057} C_VEL
LIN {X 0,Y 193.182,Z 682.025,A -85,B 0,C 180,E1 -24659.791,E2 -24659.791} C_VEL
LIN {X 0,Y 189.764,Z 694.164,A -85,B 0,C 180,E1 -24660.822,E2 -24660.822} C_VEL
LIN {X 0,Y 185.462,Z 705.864,A -85,B 0,C 180,E1 -24662.171,E2 -24662.171} C_VEL
LIN {X 0,Y 180.408,Z 716.96,A -85,B 0,C 180,E1 -24663.847,E2 -24663.847} C_VEL
LIN {X 0,Y 174.555,Z 727.689,A -85,B 0,C 180,E1 -24666.007,E2 -24666.007} C_VEL
LIN {X 0,Y 168.985,Z 736.441,A -85,B 0,C 180,E1 -24668.327,E2 -24668.327} C_VEL
LIN {X 0,Y 163.158,Z 744.395,A -85,B 0,C 180,E1 -24671.063,E2 -24671.063} C_VEL
LIN {X 0,Y 156.646,Z 752.171,A -85,B 0,C 180,E1 -24674.654,E2 -24674.654} C_VEL
LIN {X 0,Y 151.734,Z 757.318,A -85,B 0,C 180,E1 -24677.873,E2 -24677.873} C_VEL
LIN {X 0,Y 147.359,Z 761.444,A -85,B 0,C 180,E1 -24681.295,E2 -24681.295} C_VEL
LIN {X 0,Y 143.532,Z 764.632,A -85,B 0,C 180,E1 -24684.88,E2 -24684.88} C_VEL
LIN {X 0,Y 139.126,Z 767.772,A -85,B 0,C 180,E1 -24690.34,E2 -24690.34} C_VEL
LIN {X 0,Y 136.621,Z 769.071,A -85,B 0,C 180,E1 -24694.615,E2 -24694.615} C_VEL
LIN {X 0,Y 134.946,Z 769.468,A -85,B 0,C 180,E1 -24698.677,E2 -24698.677} C_VEL
LIN {X 0,Y 133.684,Z 769.092,A -85,B 0,C 180,E1 -24703.11,E2 -24703.11} C_VEL
LIN {X 0,Y 133.039,Z 767.816,A -85,B 0,C 180,E1 -24707.693,E2 -24707.693} C_VEL
LIN {X 0,Y 133.023,Z 765.529,A -85,B 0,C 180,E1 -24712.417,E2 -24712.417} C_VEL
LIN {X 0,Y 133.615,Z 762.031,A -85,B 0,C 180,E1 -24717.305,E2 -24717.305} C_VEL
LIN {X 0,Y 134.849,Z 757.024,A -85,B 0,C 180,E1 -24722.371,E2 -24722.371} C_VEL
LIN {X 0,Y 136.437,Z 751.411,A -85,B 0,C 180,E1 -24726.694,E2 -24726.694} C_VEL
LIN {X 0,Y 138.466,Z 744.759,A -85,B 0,C 180,E1 -24730.741,E2 -24730.741} C_VEL
LIN {X 0,Y 141.278,Z 736.058,A -85,B 0,C 180,E1 -24734.865,E2 -24734.865} C_VEL
LIN {X 0,Y 144.167,Z 726.717,A -85,B 0,C 180,E1 -24738.338,E2 -24738.338} C_VEL
LIN {X 0,Y 147.305,Z 716.036,A -85,B 0,C 180,E1 -24741.43,E2 -24741.43} C_VEL
LIN {X 0,Y 150.308,Z 704.307,A -85,B 0,C 180,E1 -24744.023,E2 -24744.023} C_VEL
LIN {X 0,Y 152.926,Z 692.235,A -85,B 0,C 180,E1 -24746.052,E2 -24746.052} C_VEL
LIN {X 0,Y 155.132,Z 679.275,A -85,B 0,C 180,E1 -24747.624,E2 -24747.624} C_VEL
LIN {X 0,Y 156.708,Z 666.99,A -85,B 0,C 180,E1 -24748.639,E2 -24748.639} C_VEL
LIN {X 0,Y 159.347,Z 631.129,A -85,B 0,C 180,E1 -24750.394,E2 -24750.394} C_VEL
LIN {X 0,Y 160.313,Z 616.074,A -85,B 0,C 180,E1 -24751.109,E2 -24751.109} C_VEL
LIN {X 0,Y 156.426,Z 605.055,A -85,B 0,C 180,E1 -24752.669,E2 -24752.669} C_VEL
LIN {X 0,Y 148.651,Z 588.526,A -85,B 0,C 180,E1 -24755.681,E2 -24755.681} C_VEL
LIN {X 0,Y 138.723,Z 571.727,A -85,B 0,C 180,E1 -24759.828,E2 -24759.828} C_VEL
LIN {X 0,Y 136.987,Z 569.151,A -85,B 0,C 180,E1 -24760.6,E2 -24760.6} C_VEL
LIN {X 0,Y 136.551,Z 567.462,A -85,B 0,C 180,E1 -24760.95,E2 -24760.95} C_VEL
LIN {X 0,Y 136.253,Z 567.512,A -85,B 0,C 180,E1 -24768.032,E2 -24768.032} C_VEL
LIN {X 0,Y 136.199,Z 567.483,A -85,B 0,C 180,E1 -24771.753,E2 -24771.753} C_VEL
LIN {X 0,Y 136.102,Z 567.534,A -85,B 0,C 180,E1 -24778.62,E2 -24778.62} C_VEL
LIN {X 0,Y 136.045,Z 567.537,A -85,B 0,C 180,E1 -24784.633,E2 -24784.633} C_VEL
LIN {X 0,Y 136.034,Z 567.53,A -85,B 0,C 180,E1 -24789.202,E2 -24789.202} C_VEL
LIN {X 0,Y 136.001,Z 567.541,A -85,B 0,C 180,E1 -24793.661,E2 -24793.661} C_VEL
LIN {X 0,Y 136.009,Z 567.536,A -85,B 0,C 180,E1 -24797.8,E2 -24797.8} C_VEL
LIN {X 0,Y 136.031,Z 567.522,A -85,B 0,C 180,E1 -24801.688,E2 -24801.688} C_VEL
LIN {X 0,Y 136.061,Z 567.537,A -85,B 0,C 180,E1 -24805.743,E2 -24805.743} C_VEL
LIN {X 0,Y 136.151,Z 567.504,A -85,B 0,C 180,E1 -24812.319,E2 -24812.319} C_VEL
LIN {X 0,Y 136.248,Z 567.51,A -85,B 0,C 180,E1 -24818.835,E2 -24818.835} C_VEL
LIN {X 0,Y 136.265,Z 567.5,A -85,B 0,C 180,E1 -24825.057,E2 -24825.057} C_VEL
LIN {X 0,Y 136.439,Z 567.489,A -85,B 0,C 180,E1 -24828.17,E2 -24828.17} C_VEL
LIN {X 0,Y 136.56,Z 567.464,A -85,B 0,C 180,E1 -24831.12,E2 -24831.12} C_VEL
LIN {X 0,Y 137.143,Z 567.4,A -85,B 0,C 180,E1 -24840.002,E2 -24840.002} C_VEL
LIN {X 0,Y 136.609,Z 567.469,A -85,B 0,C 180,E1 -24848.88,E2 -24848.88} C_VEL
LIN {X 0,Y 136.501,Z 567.469,A -85,B 0,C 180,E1 -24851.955,E2 -24851.955} C_VEL
LIN {X 0,Y 136.252,Z 567.513,A -85,B 0,C 180,E1 -24858.03,E2 -24858.03} C_VEL
LIN {X 0,Y 136.206,Z 567.488,A -85,B 0,C 180,E1 -24861.746,E2 -24861.746} C_VEL
LIN {X 0,Y 136.109,Z 567.527,A -85,B 0,C 180,E1 -24868.614,E2 -24868.614} C_VEL
LIN {X 0,Y 136.052,Z 567.54,A -85,B 0,C 180,E1 -24874.628,E2 -24874.628} C_VEL
LIN {X 0,Y 136.032,Z 567.569,A -85,B 0,C 180,E1 -24878.471,E2 -24878.471} C_VEL
LIN {X 0,Y 136.977,Z 570.321,A -85,B 0,C 180,E1 -24879.014,E2 -24879.014} C_VEL
LIN {X 0,Y 138.746,Z 572.776,A -85,B 0,C 180,E1 -24879.792,E2 -24879.792} C_VEL
LIN {X 0,Y 144.11,Z 581.961,A -85,B 0,C 180,E1 -24882.115,E2 -24882.115} C_VEL
LIN {X 0,Y 150.908,Z 597.326,A -85,B 0,C 180,E1 -24885.025,E2 -24885.025} C_VEL
LIN {X 0,Y 157.107,Z 614.306,A -85,B 0,C 180,E1 -24887.597,E2 -24887.597} C_VEL
LIN {X 0,Y 159.182,Z 620.794,A -85,B 0,C 180,E1 -24888.462,E2 -24888.462} C_VEL
LIN {X 0,Y 159.859,Z 628.158,A -85,B 0,C 180,E1 -24889.058,E2 -24889.058} C_VEL
LIN {X 0,Y 156.609,Z 674.108,A -85,B 0,C 180,E1 -24891.28,E2 -24891.28} C_VEL
LIN {X 0,Y 154.776,Z 687.865,A -85,B 0,C 180,E1 -24892.394,E2 -24892.394} C_VEL
LIN {X 0,Y 152.767,Z 698.773,A -85,B 0,C 180,E1 -24893.675,E2 -24893.675} C_VEL
LIN {X 0,Y 150.355,Z 710.072,A -85,B 0,C 180,E1 -24895.471,E2 -24895.471} C_VEL
LIN {X 0,Y 147.301,Z 721.776,A -85,B 0,C 180,E1 -24897.937,E2 -24897.937} C_VEL
LIN {X 0,Y 144.24,Z 732.353,A -85,B 0,C 180,E1 -24900.836,E2 -24900.836} C_VEL
LIN {X 0,Y 141.194,Z 741.873,A -85,B 0,C 180,E1 -24904.176,E2 -24904.176} C_VEL
LIN {X 0,Y 138.796,Z 749.698,A -85,B 0,C 180,E1 -24907.676,E2 -24907.676} C_VEL
LIN {X 0,Y 136.437,Z 757.317,A -85,B 0,C 180,E1 -24911.993,E2 -24911.993} C_VEL
LIN {X 0,Y 134.831,Z 763.411,A -85,B 0,C 180,E1 -24916.43,E2 -24916.43} C_VEL
LIN {X 0,Y 133.947,Z 768.2,A -85,B 0,C 180,E1 -24920.939,E2 -24920.939} C_VEL
LIN {X 0,Y 133.547,Z 771.807,A -85,B 0,C 180,E1 -24925.468,E2 -24925.468} C_VEL
LIN {X 0,Y 133.546,Z 774.689,A -85,B 0,C 180,E1 -24930.729,E2 -24930.729} C_VEL
LIN {X 0,Y 133.55,Z 776.227,A -85,B 0,C 180,E1 -24936.037,E2 -24936.037} C_VEL
LIN {X 0,Y 134.478,Z 776.487,A -85,B 0,C 180,E1 -24942.062,E2 -24942.062} C_VEL
LIN {X 0,Y 136.678,Z 775.257,A -85,B 0,C 180,E1 -24947.966,E2 -24947.966} C_VEL
LIN {X 0,Y 138.703,Z 773.766,A -85,B 0,C 180,E1 -24951.309,E2 -24951.309} C_VEL
LIN {X 0,Y 139.785,Z 772.508,A -85,B 0,C 180,E1 -24953.637,E2 -24953.637} C_VEL
LIN {X 0,Y 140.294,Z 770.028,A -85,B 0,C 180,E1 -24957.573,E2 -24957.573} C_VEL
LIN {X 0,Y 141.362,Z 767.058,A -85,B 0,C 180,E1 -24961.397,E2 -24961.397} C_VEL
LIN {X 0,Y 143.248,Z 764.838,A -85,B 0,C 180,E1 -24963.465,E2 -24963.465} C_VEL
LIN {X 0,Y 147.679,Z 760.527,A -85,B 0,C 180,E1 -24966.498,E2 -24966.498} C_VEL
LIN {X 0,Y 153.638,Z 754.212,A -85,B 0,C 180,E1 -24969.818,E2 -24969.818} C_VEL
LIN {X 0,Y 160.005,Z 746.425,A -85,B 0,C 180,E1 -24972.902,E2 -24972.902} C_VEL
LIN {X 0,Y 166.901,Z 736.892,A -85,B 0,C 180,E1 -24975.707,E2 -24975.707} C_VEL
LIN {X 0,Y 173.03,Z 727.105,A -85,B 0,C 180,E1 -24977.834,E2 -24977.834} C_VEL
LIN {X 0,Y 178.761,Z 716.199,A -85,B 0,C 180,E1 -24979.611,E2 -24979.611} C_VEL
LIN {X 0,Y 184.08,Z 704.004,A -85,B 0,C 180,E1 -24981.063,E2 -24981.063} C_VEL
LIN {X 0,Y 188.174,Z 692.041,A -85,B 0,C 180,E1 -24982.11,E2 -24982.11} C_VEL
LIN {X 0,Y 191.74,Z 678.021,A -85,B 0,C 180,E1 -24982.929,E2 -24982.929} C_VEL
LIN {X 0,Y 193.817,Z 665.095,A -85,B 0,C 180,E1 -24983.469,E2 -24983.469} C_VEL
LIN {X 0,Y 195.416,Z 651.286,A -85,B 0,C 180,E1 -24983.96,E2 -24983.96} C_VEL
LIN {X 0,Y 193.326,Z 644.825,A -85,B 0,C 180,E1 -24986.574,E2 -24986.574} C_VEL
LIN {X 0,Y 191.754,Z 640.215,A -85,B 0,C 180,E1 -24988.932,E2 -24988.932} C_VEL
LIN {X 0,Y 190.094,Z 635.875,A -85,B 0,C 180,E1 -24992.014,E2 -24992.014} C_VEL
LIN {X 0,Y 188.608,Z 631.641,A -85,B 0,C 180,E1 -24996.989,E2 -24996.989} C_VEL
LIN {X 0,Y 188.292,Z 630.932,A -85,B 0,C 180,E1 -25000.37,E2 -25000.37} C_VEL
LIN {X 0,Y 188.778,Z 631.159,A -85,B 0,C 180,E1 -25003.911,E2 -25003.911} C_VEL
LIN {X 0,Y 190.352,Z 633.903,A -85,B 0,C 180,E1 -25008.409,E2 -25008.409} C_VEL
LIN {X 0,Y 192.699,Z 638.24,A -85,B 0,C 180,E1 -25012.285,E2 -25012.285} C_VEL
LIN {X 0,Y 195.565,Z 645.577,A -85,B 0,C 180,E1 -25015.94,E2 -25015.94} C_VEL
LIN {X 0,Y 195.874,Z 646.673,A -85,B 0,C 180,E1 -25016.323,E2 -25016.323} C_VEL
LIN {X 0,Y 192.877,Z 670.029,A -85,B 0,C 180,E1 -25017.189,E2 -25017.189} C_VEL
LIN {X 0,Y 190.164,Z 682.526,A -85,B 0,C 180,E1 -25017.881,E2 -25017.881} C_VEL
LIN {X 0,Y 186.704,Z 694.306,A -85,B 0,C 180,E1 -25018.854,E2 -25018.854} C_VEL
LIN {X 0,Y 182.051,Z 706.484,A -85,B 0,C 180,E1 -25020.237,E2 -25020.237} C_VEL
LIN {X 0,Y 176.667,Z 717.795,A -85,B 0,C 180,E1 -25021.932,E2 -25021.932} C_VEL
LIN {X 0,Y 170.828,Z 727.963,A -85,B 0,C 180,E1 -25023.974,E2 -25023.974} C_VEL
LIN {X 0,Y 164.44,Z 737.386,A -85,B 0,C 180,E1 -25026.48,E2 -25026.48} C_VEL
LIN {X 0,Y 158.392,Z 745.106,A -85,B 0,C 180,E1 -25029.183,E2 -25029.183} C_VEL
LIN {X 0,Y 152.499,Z 751.741,A -85,B 0,C 180,E1 -25032.232,E2 -25032.232} C_VEL
LIN {X 0,Y 146.283,Z 757.886,A -85,B 0,C 180,E1 -25036.095,E2 -25036.095} C_VEL
LIN {X 0,Y 140.551,Z 762.773,A -85,B 0,C 180,E1 -25040.487,E2 -25040.487} C_VEL
LIN {X 0,Y 136.515,Z 765.749,A -85,B 0,C 180,E1 -25044.32,E2 -25044.32} C_VEL
LIN {X 0,Y 133.17,Z 767.878,A -85,B 0,C 180,E1 -25048.356,E2 -25048.356} C_VEL
LIN {X 0,Y 130.401,Z 769.181,A -85,B 0,C 180,E1 -25052.61,E2 -25052.61} C_VEL
LIN {X 0,Y 128.371,Z 769.682,A -85,B 0,C 180,E1 -25057.027,E2 -25057.027} C_VEL
LIN {X 0,Y 126.899,Z 769.383,A -85,B 0,C 180,E1 -25061.649,E2 -25061.649} C_VEL
LIN {X 0,Y 125.916,Z 767.649,A -85,B 0,C 180,E1 -25067.956,E2 -25067.956} C_VEL
LIN {X 0,Y 125.923,Z 765.621,A -85,B 0,C 180,E1 -25072.132,E2 -25072.132} C_VEL
LIN {X 0,Y 126.401,Z 762.706,A -85,B 0,C 180,E1 -25076.51,E2 -25076.51} C_VEL
LIN {X 0,Y 127.547,Z 757.87,A -85,B 0,C 180,E1 -25081.835,E2 -25081.835} C_VEL
LIN {X 0,Y 129.204,Z 752.073,A -85,B 0,C 180,E1 -25086.658,E2 -25086.658} C_VEL
LIN {X 0,Y 131.492,Z 744.881,A -85,B 0,C 180,E1 -25091.3,E2 -25091.3} C_VEL
LIN {X 0,Y 134.418,Z 736.154,A -85,B 0,C 180,E1 -25095.625,E2 -25095.625} C_VEL
LIN {X 0,Y 137.512,Z 726.552,A -85,B 0,C 180,E1 -25099.335,E2 -25099.335} C_VEL
LIN {X 0,Y 140.605,Z 716.468,A -85,B 0,C 180,E1 -25102.369,E2 -25102.369} C_VEL
LIN {X 0,Y 143.79,Z 704.622,A -85,B 0,C 180,E1 -25105.097,E2 -25105.097} C_VEL
LIN {X 0,Y 146.585,Z 692.228,A -85,B 0,C 180,E1 -25107.256,E2 -25107.256} C_VEL
LIN {X 0,Y 148.894,Z 679.077,A -85,B 0,C 180,E1 -25108.891,E2 -25108.891} C_VEL
LIN {X 0,Y 150.625,Z 665.71,A -85,B 0,C 180,E1 -25110.004,E2 -25110.004} C_VEL
LIN {X 0,Y 154.195,Z 617.799,A -85,B 0,C 180,E1 -25112.361,E2 -25112.361} C_VEL
LIN {X 0,Y 150.692,Z 608.042,A -85,B 0,C 180,E1 -25113.83,E2 -25113.83} C_VEL
LIN {X 0,Y 143.506,Z 592.463,A -85,B 0,C 180,E1 -25116.83,E2 -25116.83} C_VEL
LIN {X 0,Y 134.223,Z 576.664,A -85,B 0,C 180,E1 -25120.934,E2 -25120.934} C_VEL
LIN {X 0,Y 131.583,Z 572.603,A -85,B 0,C 180,E1 -25122.197,E2 -25122.197} C_VEL
LIN {X 0,Y 129.845,Z 570.26,A -85,B 0,C 180,E1 -25123.034,E2 -25123.034} C_VEL
LIN {X 0,Y 129.294,Z 568.357,A -85,B 0,C 180,E1 -25123.442,E2 -25123.442} C_VEL
LIN {X 0,Y 129.161,Z 568.383,A -85,B 0,C 180,E1 -25129.06,E2 -25129.06} C_VEL
LIN {X 0,Y 129.109,Z 568.363,A -85,B 0,C 180,E1 -25132.403,E2 -25132.403} C_VEL
LIN {X 0,Y 129.032,Z 568.4,A -85,B 0,C 180,E1 -25135.837,E2 -25135.837} C_VEL
LIN {X 0,Y 129.018,Z 568.416,A -85,B 0,C 180,E1 -25139.362,E2 -25139.362} C_VEL
LIN {X 0,Y 128.962,Z 568.421,A -85,B 0,C 180,E1 -25145.173,E2 -25145.173} C_VEL
LIN {X 0,Y 128.937,Z 568.407,A -85,B 0,C 180,E1 -25150.856,E2 -25150.856} C_VEL
LIN {X 0,Y 128.926,Z 568.426,A -85,B 0,C 180,E1 -25155.132,E2 -25155.132} C_VEL
LIN {X 0,Y 128.947,Z 568.402,A -85,B 0,C 180,E1 -25159.74,E2 -25159.74} C_VEL
LIN {X 0,Y 128.965,Z 568.419,A -85,B 0,C 180,E1 -25164.836,E2 -25164.836} C_VEL
LIN {X 0,Y 129.023,Z 568.39,A -85,B 0,C 180,E1 -25170.646,E2 -25170.646} C_VEL
LIN {X 0,Y 129.034,Z 568.402,A -85,B 0,C 180,E1 -25174.17,E2 -25174.17} C_VEL
LIN {X 0,Y 129.114,Z 568.4,A -85,B 0,C 180,E1 -25177.732,E2 -25177.732} C_VEL
LIN {X 0,Y 129.184,Z 568.373,A -85,B 0,C 180,E1 -25184.217,E2 -25184.217} C_VEL
LIN {X 0,Y 129.384,Z 568.368,A -85,B 0,C 180,E1 -25187.907,E2 -25187.907} C_VEL
LIN {X 0,Y 129.483,Z 568.349,A -85,B 0,C 180,E1 -25190.63,E2 -25190.63} C_VEL
LIN {X 0,Y 130.098,Z 568.278,A -85,B 0,C 180,E1 -25200.002,E2 -25200.002} C_VEL
LIN {X 0,Y 129.533,Z 568.351,A -85,B 0,C 180,E1 -25209.369,E2 -25209.369} C_VEL
LIN {X 0,Y 129.403,Z 568.351,A -85,B 0,C 180,E1 -25212.549,E2 -25212.549} C_VEL
LIN {X 0,Y 129.163,Z 568.391,A -85,B 0,C 180,E1 -25219.056,E2 -25219.056} C_VEL
LIN {X 0,Y 129.118,Z 568.362,A -85,B 0,C 180,E1 -25222.398,E2 -25222.398} C_VEL
LIN {X 0,Y 129.037,Z 568.375,A -85,B 0,C 180,E1 -25225.833,E2 -25225.833} C_VEL
LIN {X 0,Y 129.027,Z 568.412,A -85,B 0,C 180,E1 -25229.357,E2 -25229.357} C_VEL
LIN {X 0,Y 128.957,Z 568.42,A -85,B 0,C 180,E1 -25235.774,E2 -25235.774} C_VEL
LIN {X 0,Y 128.942,Z 568.427,A -85,B 0,C 180,E1 -25235.976,E2 -25235.976} C_VEL
LIN {X 0,Y 129.841,Z 571.109,A -85,B 0,C 180,E1 -25236.544,E2 -25236.544} C_VEL
LIN {X 0,Y 131.777,Z 573.685,A -85,B 0,C 180,E1 -25237.47,E2 -25237.47} C_VEL
LIN {X 0,Y 138.419,Z 584.735,A -85,B 0,C 180,E1 -25240.602,E2 -25240.602} C_VEL
LIN {X 0,Y 144.551,Z 598.45,A -85,B 0,C 180,E1 -25243.42,E2 -25243.42} C_VEL
LIN {X 0,Y 149.67,Z 612.091,A -85,B 0,C 180,E1 -25245.71,E2 -25245.71} C_VEL
LIN {X 0,Y 153.182,Z 622.549,A -85,B 0,C 180,E1 -25247.231,E2 -25247.231} C_VEL
LIN {X 0,Y 153.721,Z 629.106,A -85,B 0,C 180,E1 -25247.774,E2 -25247.774} C_VEL
LIN {X 0,Y 150.386,Z 673.974,A -85,B 0,C 180,E1 -25250.011,E2 -25250.011} C_VEL
LIN {X 0,Y 148.497,Z 687.681,A -85,B 0,C 180,E1 -25251.16,E2 -25251.16} C_VEL
LIN {X 0,Y 146.191,Z 699.647,A -85,B 0,C 180,E1 -25252.627,E2 -25252.627} C_VEL
LIN {X 0,Y 143.683,Z 710.642,A -85,B 0,C 180,E1 -25254.485,E2 -25254.485} C_VEL
LIN {X 0,Y 140.538,Z 722.182,A -85,B 0,C 180,E1 -25257.05,E2 -25257.05} C_VEL
LIN {X 0,Y 137.374,Z 732.645,A -85,B 0,C 180,E1 -25260.075,E2 -25260.075} C_VEL
LIN {X 0,Y 134.245,Z 742.039,A -85,B 0,C 180,E1 -25263.573,E2 -25263.573} C_VEL
LIN {X 0,Y 131.753,Z 749.79,A -85,B 0,C 180,E1 -25267.244,E2 -25267.244} C_VEL
LIN {X 0,Y 129.325,Z 757.346,A -85,B 0,C 180,E1 -25271.787,E2 -25271.787} C_VEL
LIN {X 0,Y 127.524,Z 764.288,A -85,B 0,C 180,E1 -25277.26,E2 -25277.26} C_VEL
LIN {X 0,Y 126.723,Z 768.816,A -85,B 0,C 180,E1 -25282.026,E2 -25282.026} C_VEL
LIN {X 0,Y 126.452,Z 772.203,A -85,B 0,C 180,E1 -25286.809,E2 -25286.809} C_VEL
LIN {X 0,Y 126.51,Z 774.015,A -85,B 0,C 180,E1 -25290.353,E2 -25290.353} C_VEL
LIN {X 0,Y 126.501,Z 775.892,A -85,B 0,C 180,E1 -25296.375,E2 -25296.375} C_VEL
LIN {X 0,Y 126.856,Z 776.303,A -85,B 0,C 180,E1 -25299.563,E2 -25299.563} C_VEL
LIN {X 0,Y 128.56,Z 775.952,A -85,B 0,C 180,E1 -25305.858,E2 -25305.858} C_VEL
LIN {X 0,Y 131.753,Z 774.125,A -85,B 0,C 180,E1 -25311.92,E2 -25311.92} C_VEL
LIN {X 0,Y 133.99,Z 772.61,A -85,B 0,C 180,E1 -25314.805,E2 -25314.805} C_VEL
LIN {X 0,Y 139.322,Z 768.348,A -85,B 0,C 180,E1 -25320.289,E2 -25320.289} C_VEL
LIN {X 0,Y 143.248,Z 764.838,A -85,B 0,C 180,E1 -25323.465,E2 -25323.465} C_VEL
LIN {X 0,Y 145.298,Z 762.425,A -85,B 0,C 180,E1 -25325.453,E2 -25325.453} C_VEL
LIN {X 0,Y 147.459,Z 758.271,A -85,B 0,C 180,E1 -25328.889,E2 -25328.889} C_VEL
LIN {X 0,Y 150.049,Z 753.596,A -85,B 0,C 180,E1 -25332.093,E2 -25332.093} C_VEL
LIN {X 0,Y 152.653,Z 750.323,A -85,B 0,C 180,E1 -25333.665,E2 -25333.665} C_VEL
LIN {X 0,Y 159.718,Z 741.709,A -85,B 0,C 180,E1 -25336.55,E2 -25336.55} C_VEL
LIN {X 0,Y 165.891,Z 732.995,A -85,B 0,C 180,E1 -25338.756,E2 -25338.756} C_VEL
LIN {X 0,Y 172.394,Z 722.35,A -85,B 0,C 180,E1 -25340.76,E2 -25340.76} C_VEL
LIN {X 0,Y 177.75,Z 711.857,A -85,B 0,C 180,E1 -25342.252,E2 -25342.252} C_VEL
LIN {X 0,Y 182.597,Z 700.344,A -85,B 0,C 180,E1 -25343.456,E2 -25343.456} C_VEL
LIN {X 0,Y 186.817,Z 687.562,A -85,B 0,C 180,E1 -25344.42,E2 -25344.42} C_VEL
LIN {X 0,Y 189.867,Z 674.616,A -85,B 0,C 180,E1 -25345.081,E2 -25345.081} C_VEL
LIN {X 0,Y 192.603,Z 654.9,A -85,B 0,C 180,E1 -25345.786,E2 -25345.786} C_VEL
LIN {X 0,Y 190.751,Z 648.71,A -85,B 0,C 180,E1 -25348.554,E2 -25348.554} C_VEL
LIN {X 0,Y 189.527,Z 645.178,A -85,B 0,C 180,E1 -25350.737,E2 -25350.737} C_VEL
LIN {X 0,Y 188.626,Z 642.321,A -85,B 0,C 180,E1 -25352.842,E2 -25352.842} C_VEL
LIN {X 0,Y 187.469,Z 638.564,A -85,B 0,C 180,E1 -25357.363,E2 -25357.363} C_VEL
LIN {X 0,Y 187.221,Z 637.965,A -85,B 0,C 180,E1 -25360.253,E2 -25360.253} C_VEL
LIN {X 0,Y 187.649,Z 638.107,A -85,B 0,C 180,E1 -25363.643,E2 -25363.643} C_VEL
LIN {X 0,Y 189.033,Z 640.772,A -85,B 0,C 180,E1 -25367.966,E2 -25367.966} C_VEL
LIN {X 0,Y 191.179,Z 645.061,A -85,B 0,C 180,E1 -25371.788,E2 -25371.788} C_VEL
LIN {X 0,Y 193.047,Z 650.445,A -85,B 0,C 180,E1 -25374.493,E2 -25374.493} C_VEL
LIN {X 0,Y 190.415,Z 669.967,A -85,B 0,C 180,E1 -25375.191,E2 -25375.191} C_VEL
LIN {X 0,Y 187.752,Z 682.003,A -85,B 0,C 180,E1 -25375.823,E2 -25375.823} C_VEL
LIN {X 0,Y 183.805,Z 694.973,A -85,B 0,C 180,E1 -25376.867,E2 -25376.867} C_VEL
LIN {X 0,Y 178.956,Z 707.036,A -85,B 0,C 180,E1 -25378.213,E2 -25378.213} C_VEL
LIN {X 0,Y 173.937,Z 717.116,A -85,B 0,C 180,E1 -25379.673,E2 -25379.673} C_VEL
LIN {X 0,Y 167.775,Z 727.581,A -85,B 0,C 180,E1 -25381.688,E2 -25381.688} C_VEL
LIN {X 0,Y 161.03,Z 737.183,A -85,B 0,C 180,E1 -25384.169,E2 -25384.169} C_VEL
LIN {X 0,Y 153.632,Z 746.141,A -85,B 0,C 180,E1 -25387.285,E2 -25387.285} C_VEL
LIN {X 0,Y 147.586,Z 752.438,A -85,B 0,C 180,E1 -25390.264,E2 -25390.264} C_VEL
LIN {X 0,Y 140.557,Z 758.812,A -85,B 0,C 180,E1 -25394.476,E2 -25394.476} C_VEL
LIN {X 0,Y 134.066,Z 763.862,A -85,B 0,C 180,E1 -25399.349,E2 -25399.349} C_VEL
LIN {X 0,Y 129.963,Z 766.508,A -85,B 0,C 180,E1 -25403.187,E2 -25403.187} C_VEL
LIN {X 0,Y 126.515,Z 768.391,A -85,B 0,C 180,E1 -25407.287,E2 -25407.287} C_VEL
LIN {X 0,Y 123.689,Z 769.538,A -85,B 0,C 180,E1 -25411.547,E2 -25411.547} C_VEL
LIN {X 0,Y 121.587,Z 769.917,A -85,B 0,C 180,E1 -25415.988,E2 -25415.988} C_VEL
LIN {X 0,Y 120.075,Z 769.599,A -85,B 0,C 180,E1 -25420.465,E2 -25420.465} C_VEL
LIN {X 0,Y 119.104,Z 768.571,A -85,B 0,C 180,E1 -25425.077,E2 -25425.077} C_VEL
LIN {X 0,Y 118.768,Z 766.503,A -85,B 0,C 180,E1 -25430.285,E2 -25430.285} C_VEL
LIN {X 0,Y 119.159,Z 763.318,A -85,B 0,C 180,E1 -25435.659,E2 -25435.659} C_VEL
LIN {X 0,Y 120.244,Z 758.689,A -85,B 0,C 180,E1 -25441.245,E2 -25441.245} C_VEL
LIN {X 0,Y 122.137,Z 752.223,A -85,B 0,C 180,E1 -25447.02,E2 -25447.02} C_VEL
LIN {X 0,Y 124.33,Z 745.594,A -85,B 0,C 180,E1 -25451.556,E2 -25451.556} C_VEL
LIN {X 0,Y 126.928,Z 738.167,A -85,B 0,C 180,E1 -25455.577,E2 -25455.577} C_VEL
LIN {X 0,Y 130.147,Z 728.7,A -85,B 0,C 180,E1 -25459.588,E2 -25459.588} C_VEL
LIN {X 0,Y 133.713,Z 717.657,A -85,B 0,C 180,E1 -25463.176,E2 -25463.176} C_VEL
LIN {X 0,Y 136.938,Z 706.405,A -85,B 0,C 180,E1 -25465.958,E2 -25465.958} C_VEL
LIN {X 0,Y 139.878,Z 694.001,A -85,B 0,C 180,E1 -25468.274,E2 -25468.274} C_VEL
LIN {X 0,Y 142.052,Z 683.145,A -85,B 0,C 180,E1 -25469.767,E2 -25469.767} C_VEL
LIN {X 0,Y 143.855,Z 670.508,A -85,B 0,C 180,E1 -25471.04,E2 -25471.04} C_VEL
LIN {X 0,Y 145.391,Z 655.322,A -85,B 0,C 180,E1 -25471.925,E2 -25471.925} C_VEL
LIN {X 0,Y 148.038,Z 619.437,A -85,B 0,C 180,E1 -25473.718,E2 -25473.718} C_VEL
LIN {X 0,Y 145.286,Z 611.579,A -85,B 0,C 180,E1 -25474.973,E2 -25474.973} C_VEL
LIN {X 0,Y 138.57,Z 596.733,A -85,B 0,C 180,E1 -25477.958,E2 -25477.958} C_VEL
LIN {X 0,Y 129.604,Z 581.28,A -85,B 0,C 180,E1 -25482.19,E2 -25482.19} C_VEL
LIN {X 0,Y 126.947,Z 577.32,A -85,B 0,C 180,E1 -25483.537,E2 -25483.537} C_VEL
LIN {X 0,Y 124.523,Z 573.671,A -85,B 0,C 180,E1 -25484.844,E2 -25484.844} C_VEL
LIN {X 0,Y 122.732,Z 571.275,A -85,B 0,C 180,E1 -25485.827,E2 -25485.827} C_VEL
LIN {X 0,Y 122.147,Z 569.27,A -85,B 0,C 180,E1 -25486.314,E2 -25486.314} C_VEL
LIN {X 0,Y 122.029,Z 569.244,A -85,B 0,C 180,E1 -25492.86,E2 -25492.86} C_VEL
LIN {X 0,Y 121.943,Z 569.295,A -85,B 0,C 180,E1 -25497.461,E2 -25497.461} C_VEL
LIN {X 0,Y 121.901,Z 569.291,A -85,B 0,C 180,E1 -25501.262,E2 -25501.262} C_VEL
LIN {X 0,Y 121.887,Z 569.305,A -85,B 0,C 180,E1 -25506.176,E2 -25506.176} C_VEL
LIN {X 0,Y 121.876,Z 569.287,A -85,B 0,C 180,E1 -25511.443,E2 -25511.443} C_VEL
LIN {X 0,Y 121.877,Z 569.289,A -85,B 0,C 180,E1 -25518.566,E2 -25518.566} C_VEL
LIN {X 0,Y 121.917,Z 569.297,A -85,B 0,C 180,E1 -25524.8,E2 -25524.8} C_VEL
LIN {X 0,Y 121.933,Z 569.276,A -85,B 0,C 180,E1 -25529.843,E2 -25529.843} C_VEL
LIN {X 0,Y 121.989,Z 569.289,A -85,B 0,C 180,E1 -25536.218,E2 -25536.218} C_VEL
LIN {X 0,Y 122.035,Z 569.273,A -85,B 0,C 180,E1 -25539.787,E2 -25539.787} C_VEL
LIN {X 0,Y 122.244,Z 569.255,A -85,B 0,C 180,E1 -25546.707,E2 -25546.707} C_VEL
LIN {X 0,Y 122.415,Z 569.231,A -85,B 0,C 180,E1 -25550.084,E2 -25550.084} C_VEL
LIN {X 0,Y 122.607,Z 569.206,A -85,B 0,C 180,E1 -25556.716,E2 -25556.716} C_VEL
LIN {X 0,Y 123.051,Z 569.156,A -85,B 0,C 180,E1 -25560.002,E2 -25560.002} C_VEL
LIN {X 0,Y 122.461,Z 569.224,A -85,B 0,C 180,E1 -25566.593,E2 -25566.593} C_VEL
LIN {X 0,Y 122.461,Z 569.229,A -85,B 0,C 180,E1 -25569.916,E2 -25569.916} C_VEL
LIN {X 0,Y 122.272,Z 569.239,A -85,B 0,C 180,E1 -25573.294,E2 -25573.294} C_VEL
LIN {X 0,Y 122.055,Z 569.264,A -85,B 0,C 180,E1 -25580.213,E2 -25580.213} C_VEL
LIN {X 0,Y 121.992,Z 569.242,A -85,B 0,C 180,E1 -25583.785,E2 -25583.785} C_VEL
LIN {X 0,Y 121.937,Z 569.296,A -85,B 0,C 180,E1 -25590.16,E2 -25590.16} C_VEL
LIN {X 0,Y 121.963,Z 569.382,A -85,B 0,C 180,E1 -25593.193,E2 -25593.193} C_VEL
LIN {X 0,Y 122.797,Z 571.914,A -85,B 0,C 180,E1 -25593.797,E2 -25593.797} C_VEL
LIN {X 0,Y 124.765,Z 574.519,A -85,B 0,C 180,E1 -25594.865,E2 -25594.865} C_VEL
LIN {X 0,Y 126.961,Z 577.954,A -85,B 0,C 180,E1 -25596.044,E2 -25596.044} C_VEL
LIN {X 0,Y 133.472,Z 588.761,A -85,B 0,C 180,E1 -25599.311,E2 -25599.311} C_VEL
LIN {X 0,Y 139.608,Z 602.865,A -85,B 0,C 180,E1 -25602.325,E2 -25602.325} C_VEL
LIN {X 0,Y 144.416,Z 616.114,A -85,B 0,C 180,E1 -25604.638,E2 -25604.638} C_VEL
LIN {X 0,Y 147.242,Z 624.825,A -85,B 0,C 180,E1 -25605.969,E2 -25605.969} C_VEL
LIN {X 0,Y 147.653,Z 629.617,A -85,B 0,C 180,E1 -25606.396,E2 -25606.396} C_VEL
LIN {X 0,Y 144.127,Z 674.437,A -85,B 0,C 180,E1 -25608.709,E2 -25608.709} C_VEL
LIN {X 0,Y 142.166,Z 687.93,A -85,B 0,C 180,E1 -25609.889,E2 -25609.889} C_VEL
LIN {X 0,Y 139.687,Z 700.274,A -85,B 0,C 180,E1 -25611.488,E2 -25611.488} C_VEL
LIN {X 0,Y 136.631,Z 712.64,A -85,B 0,C 180,E1 -25613.729,E2 -25613.729} C_VEL
LIN {X 0,Y 133.437,Z 723.803,A -85,B 0,C 180,E1 -25616.42,E2 -25616.42} C_VEL
LIN {X 0,Y 130.395,Z 733.283,A -85,B 0,C 180,E1 -25619.376,E2 -25619.376} C_VEL
LIN {X 0,Y 127.32,Z 742.194,A -85,B 0,C 180,E1 -25622.912,E2 -25622.912} C_VEL
LIN {X 0,Y 124.275,Z 751.25,A -85,B 0,C 180,E1 -25627.555,E2 -25627.555} C_VEL
LIN {X 0,Y 121.856,Z 758.494,A -85,B 0,C 180,E1 -25632.37,E2 -25632.37} C_VEL
LIN {X 0,Y 120.566,Z 763.382,A -85,B 0,C 180,E1 -25636.512,E2 -25636.512} C_VEL
LIN {X 0,Y 119.687,Z 768.082,A -85,B 0,C 180,E1 -25641.554,E2 -25641.554} C_VEL
LIN {X 0,Y 119.369,Z 771.599,A -85,B 0,C 180,E1 -25646.62,E2 -25646.62} C_VEL
LIN {X 0,Y 119.449,Z 773.353,A -85,B 0,C 180,E1 -25649.995,E2 -25649.995} C_VEL
LIN {X 0,Y 119.307,Z 774.626,A -85,B 0,C 180,E1 -25653.372,E2 -25653.372} C_VEL
LIN {X 0,Y 119.44,Z 775.509,A -85,B 0,C 180,E1 -25656.753,E2 -25656.753} C_VEL
LIN {X 0,Y 120.57,Z 776.131,A -85,B 0,C 180,E1 -25663.478,E2 -25663.478} C_VEL
LIN {X 0,Y 123.19,Z 775.188,A -85,B 0,C 180,E1 -25670.012,E2 -25670.012} C_VEL
LIN {X 0,Y 127.586,Z 772.77,A -85,B 0,C 180,E1 -25676.142,E2 -25676.142} C_VEL
LIN {X 0,Y 131.721,Z 769.89,A -85,B 0,C 180,E1 -25680.451,E2 -25680.451} C_VEL
LIN {X 0,Y 137.245,Z 765.489,A -85,B 0,C 180,E1 -25684.98,E2 -25684.98} C_VEL
LIN {X 0,Y 142.057,Z 761.159,A -85,B 0,C 180,E1 -25688.195,E2 -25688.195} C_VEL
LIN {X 0,Y 149.366,Z 753.98,A -85,B 0,C 180,E1 -25692.1,E2 -25692.1} C_VEL
LIN {X 0,Y 152.653,Z 750.323,A -85,B 0,C 180,E1 -25693.665,E2 -25693.665} C_VEL
LIN {X 0,Y 155.341,Z 746.9,A -85,B 0,C 180,E1 -25695.157,E2 -25695.157} C_VEL
LIN {X 0,Y 158.508,Z 741.201,A -85,B 0,C 180,E1 -25697.895,E2 -25697.895} C_VEL
LIN {X 0,Y 161.672,Z 734.955,A -85,B 0,C 180,E1 -25700.394,E2 -25700.394} C_VEL
LIN {X 0,Y 164.235,Z 730.683,A -85,B 0,C 180,E1 -25701.495,E2 -25701.495} C_VEL
LIN {X 0,Y 170.819,Z 719.92,A -85,B 0,C 180,E1 -25703.343,E2 -25703.343} C_VEL
LIN {X 0,Y 176.432,Z 708.91,A -85,B 0,C 180,E1 -25704.739,E2 -25704.739} C_VEL
LIN {X 0,Y 181.249,Z 697.239,A -85,B 0,C 180,E1 -25705.828,E2 -25705.828} C_VEL
LIN {X 0,Y 185.288,Z 684.461,A -85,B 0,C 180,E1 -25706.65,E2 -25706.65} C_VEL
LIN {X 0,Y 188.308,Z 670.683,A -85,B 0,C 180,E1 -25707.292,E2 -25707.292} C_VEL
LIN {X 0,Y 189.951,Z 658.632,A -85,B 0,C 180,E1 -25707.715,E2 -25707.715} C_VEL
LIN {X 0,Y 188.648,Z 653.698,A -85,B 0,C 180,E1 -25710.142,E2 -25710.142} C_VEL
LIN {X 0,Y 187.253,Z 648.912,A -85,B 0,C 180,E1 -25713.528,E2 -25713.528} C_VEL
LIN {X 0,Y 186.324,Z 645.467,A -85,B 0,C 180,E1 -25717.839,E2 -25717.839} C_VEL
LIN {X 0,Y 186.163,Z 644.972,A -85,B 0,C 180,E1 -25720.688,E2 -25720.688} C_VEL
LIN {X 0,Y 186.546,Z 645.163,A -85,B 0,C 180,E1 -25723.544,E2 -25723.544} C_VEL
LIN {X 0,Y 187.721,Z 647.602,A -85,B 0,C 180,E1 -25727.497,E2 -25727.497} C_VEL
LIN {X 0,Y 189.475,Z 651.433,A -85,B 0,C 180,E1 -25730.962,E2 -25730.962} C_VEL
LIN {X 0,Y 190.414,Z 654.621,A -85,B 0,C 180,E1 -25732.609,E2 -25732.609} C_VEL
LIN {X 0,Y 187.874,Z 671.739,A -85,B 0,C 180,E1 -25733.221,E2 -25733.221} C_VEL
LIN {X 0,Y 185.016,Z 683.722,A -85,B 0,C 180,E1 -25733.865,E2 -25733.865} C_VEL
LIN {X 0,Y 181.381,Z 695.051,A -85,B 0,C 180,E1 -25734.758,E2 -25734.758} C_VEL
LIN {X 0,Y 176.091,Z 707.733,A -85,B 0,C 180,E1 -25736.125,E2 -25736.125} C_VEL
LIN {X 0,Y 170.56,Z 718.349,A -85,B 0,C 180,E1 -25737.637,E2 -25737.637} C_VEL
LIN {X 0,Y 163.871,Z 728.968,A -85,B 0,C 180,E1 -25739.704,E2 -25739.704} C_VEL
LIN {X 0,Y 156.691,Z 738.524,A -85,B 0,C 180,E1 -25742.206,E2 -25742.206} C_VEL
LIN {X 0,Y 149.882,Z 746.28,A -85,B 0,C 180,E1 -25744.92,E2 -25744.92} C_VEL
LIN {X 0,Y 142.127,Z 753.804,A -85,B 0,C 180,E1 -25748.546,E2 -25748.546} C_VEL
LIN {X 0,Y 134.954,Z 759.793,A -85,B 0,C 180,E1 -25752.72,E2 -25752.72} C_VEL
LIN {X 0,Y 128.54,Z 764.305,A -85,B 0,C 180,E1 -25757.323,E2 -25757.323} C_VEL
LIN {X 0,Y 125.96,Z 765.888,A -85,B 0,C 180,E1 -25759.557,E2 -25759.557} C_VEL
LIN {X 0,Y 121.77,Z 768.099,A -85,B 0,C 180,E1 -25763.827,E2 -25763.827} C_VEL
LIN {X 0,Y 118.286,Z 769.495,A -85,B 0,C 180,E1 -25768.378,E2 -25768.378} C_VEL
LIN {X 0,Y 115.531,Z 770.115,A -85,B 0,C 180,E1 -25773.193,E2 -25773.193} C_VEL
LIN {X 0,Y 113.553,Z 769.948,A -85,B 0,C 180,E1 -25778.235,E2 -25778.235} C_VEL
LIN {X 0,Y 112.238,Z 768.912,A -85,B 0,C 180,E1 -25783.532,E2 -25783.532} C_VEL
LIN {X 0,Y 111.683,Z 766.924,A -85,B 0,C 180,E1 -25789.034,E2 -25789.034} C_VEL
LIN {X 0,Y 112.051,Z 763.254,A -85,B 0,C 180,E1 -25795.64,E2 -25795.64} C_VEL
LIN {X 0,Y 112.952,Z 759.449,A -85,B 0,C 180,E1 -25800.582,E2 -25800.582} C_VEL
LIN {X 0,Y 114.783,Z 753.176,A -85,B 0,C 180,E1 -25806.693,E2 -25806.693} C_VEL
LIN {X 0,Y 117.1,Z 746.531,A -85,B 0,C 180,E1 -25811.639,E2 -25811.639} C_VEL
LIN {X 0,Y 120.094,Z 738.199,A -85,B 0,C 180,E1 -25816.467,E2 -25816.467} C_VEL
LIN {X 0,Y 123.378,Z 728.951,A -85,B 0,C 180,E1 -25820.579,E2 -25820.579} C_VEL
LIN {X 0,Y 127.119,Z 717.882,A -85,B 0,C 180,E1 -25824.346,E2 -25824.346} C_VEL
LIN {X 0,Y 130.572,Z 706.436,A -85,B 0,C 180,E1 -25827.28,E2 -25827.28} C_VEL
LIN {X 0,Y 133.815,Z 693.25,A -85,B 0,C 180,E1 -25829.806,E2 -25829.806} C_VEL
LIN {X 0,Y 136.302,Z 680.59,A -85,B 0,C 180,E1 -25831.528,E2 -25831.528} C_VEL
LIN {X 0,Y 138.147,Z 667.923,A -85,B 0,C 180,E1 -25832.692,E2 -25832.692} C_VEL
LIN {X 0,Y 140.483,Z 640.358,A -85,B 0,C 180,E1 -25834.205,E2 -25834.205} C_VEL
LIN {X 0,Y 141.945,Z 620.819,A -85,B 0,C 180,E1 -25835.219,E2 -25835.219} C_VEL
LIN {X 0,Y 139.438,Z 614.045,A -85,B 0,C 180,E1 -25836.407,E2 -25836.407} C_VEL
LIN {X 0,Y 133.434,Z 600.534,A -85,B 0,C 180,E1 -25839.271,E2 -25839.271} C_VEL
LIN {X 0,Y 125.018,Z 585.863,A -85,B 0,C 180,E1 -25843.542,E2 -25843.542} C_VEL
LIN {X 0,Y 120.423,Z 578.948,A -85,B 0,C 180,E1 -25846.101,E2 -25846.101} C_VEL
LIN {X 0,Y 118.239,Z 575.613,A -85,B 0,C 180,E1 -25847.433,E2 -25847.433} C_VEL
LIN {X 0,Y 115.637,Z 572.344,A -85,B 0,C 180,E1 -25849.012,E2 -25849.012} C_VEL
LIN {X 0,Y 114.993,Z 570.136,A -85,B 0,C 180,E1 -25849.645,E2 -25849.645} C_VEL
LIN {X 0,Y 114.869,Z 570.154,A -85,B 0,C 180,E1 -25855.364,E2 -25855.364} C_VEL
LIN {X 0,Y 114.858,Z 570.168,A -85,B 0,C 180,E1 -25861.062,E2 -25861.062} C_VEL
LIN {X 0,Y 114.783,Z 570.186,A -85,B 0,C 180,E1 -25867.761,E2 -25867.761} C_VEL
LIN {X 0,Y 114.791,Z 570.176,A -85,B 0,C 180,E1 -25872.721,E2 -25872.721} C_VEL
LIN {X 0,Y 114.799,Z 570.178,A -85,B 0,C 180,E1 -25877.671,E2 -25877.671} C_VEL
LIN {X 0,Y 114.793,Z 570.173,A -85,B 0,C 180,E1 -25882.748,E2 -25882.748} C_VEL
LIN {X 0,Y 114.862,Z 570.163,A -85,B 0,C 180,E1 -25888.947,E2 -25888.947} C_VEL
LIN {X 0,Y 114.954,Z 570.165,A -85,B 0,C 180,E1 -25896.512,E2 -25896.512} C_VEL
LIN {X 0,Y 115.002,Z 570.132,A -85,B 0,C 180,E1 -25902.21,E2 -25902.21} C_VEL
LIN {X 0,Y 115.264,Z 570.125,A -85,B 0,C 180,E1 -25907.33,E2 -25907.33} C_VEL
LIN {X 0,Y 115.373,Z 570.09,A -85,B 0,C 180,E1 -25913.004,E2 -25913.004} C_VEL
LIN {X 0,Y 116.003,Z 570.033,A -85,B 0,C 180,E1 -25920.002,E2 -25920.002} C_VEL
LIN {X 0,Y 115.403,Z 570.106,A -85,B 0,C 180,E1 -25926.998,E2 -25926.998} C_VEL
LIN {X 0,Y 115.295,Z 570.107,A -85,B 0,C 180,E1 -25932.74,E2 -25932.74} C_VEL
LIN {X 0,Y 115.022,Z 570.159,A -85,B 0,C 180,E1 -25937.79,E2 -25937.79} C_VEL
LIN {X 0,Y 114.957,Z 570.117,A -85,B 0,C 180,E1 -25943.491,E2 -25943.491} C_VEL
LIN {X 0,Y 114.928,Z 570.362,A -85,B 0,C 180,E1 -25949.915,E2 -25949.915} C_VEL
LIN {X 0,Y 115.896,Z 573.014,A -85,B 0,C 180,E1 -25950.685,E2 -25950.685} C_VEL
LIN {X 0,Y 117.946,Z 575.477,A -85,B 0,C 180,E1 -25951.944,E2 -25951.944} C_VEL
LIN {X 0,Y 120.102,Z 578.863,A -85,B 0,C 180,E1 -25953.273,E2 -25953.273} C_VEL
LIN {X 0,Y 127.29,Z 590.653,A -85,B 0,C 180,E1 -25957.269,E2 -25957.269} C_VEL
LIN {X 0,Y 130.403,Z 596.814,A -85,B 0,C 180,E1 -25958.92,E2 -25958.92} C_VEL
LIN {X 0,Y 136.258,Z 611.439,A -85,B 0,C 180,E1 -25961.985,E2 -25961.985} C_VEL
LIN {X 0,Y 141.371,Z 627.227,A -85,B 0,C 180,E1 -25964.612,E2 -25964.612} C_VEL
LIN {X 0,Y 141.654,Z 630.249,A -85,B 0,C 180,E1 -25964.906,E2 -25964.906} C_VEL
LIN {X 0,Y 138.078,Z 673.917,A -85,B 0,C 180,E1 -25967.22,E2 -25967.22} C_VEL
LIN {X 0,Y 135.912,Z 688.18,A -85,B 0,C 180,E1 -25968.501,E2 -25968.501} C_VEL
LIN {X 0,Y 133.247,Z 700.875,A -85,B 0,C 180,E1 -25970.238,E2 -25970.238} C_VEL
LIN {X 0,Y 130.071,Z 713.083,A -85,B 0,C 180,E1 -25972.56,E2 -25972.56} C_VEL
LIN {X 0,Y 126.754,Z 724.112,A -85,B 0,C 180,E1 -25975.361,E2 -25975.361} C_VEL
LIN {X 0,Y 123.024,Z 735.045,A -85,B 0,C 180,E1 -25979.054,E2 -25979.054} C_VEL
LIN {X 0,Y 119.83,Z 743.944,A -85,B 0,C 180,E1 -25982.96,E2 -25982.96} C_VEL
LIN {X 0,Y 117.231,Z 751.291,A -85,B 0,C 180,E1 -25987.061,E2 -25987.061} C_VEL
LIN {X 0,Y 114.754,Z 758.464,A -85,B 0,C 180,E1 -25992.163,E2 -25992.163} C_VEL
LIN {X 0,Y 113.267,Z 764.171,A -85,B 0,C 180,E1 -25997.452,E2 -25997.452} C_VEL
LIN {X 0,Y 112.472,Z 768.611,A -85,B 0,C 180,E1 -26002.816,E2 -26002.816} C_VEL
LIN {X 0,Y 112.315,Z 770.929,A -85,B 0,C 180,E1 -26006.407,E2 -26006.407} C_VEL
LIN {X 0,Y 112.367,Z 772.794,A -85,B 0,C 180,E1 -26009.995,E2 -26009.995} C_VEL
LIN {X 0,Y 112.237,Z 774.173,A -85,B 0,C 180,E1 -26013.585,E2 -26013.585} C_VEL
LIN {X 0,Y 112.402,Z 775.126,A -85,B 0,C 180,E1 -26017.179,E2 -26017.179} C_VEL
LIN {X 0,Y 113.663,Z 775.895,A -85,B 0,C 180,E1 -26024.314,E2 -26024.314} C_VEL
LIN {X 0,Y 116.517,Z 775.168,A -85,B 0,C 180,E1 -26031.212,E2 -26031.212} C_VEL
LIN {X 0,Y 121.243,Z 772.903,A -85,B 0,C 180,E1 -26037.623,E2 -26037.623} C_VEL
LIN {X 0,Y 127.284,Z 769.093,A -85,B 0,C 180,E1 -26043.509,E2 -26043.509} C_VEL
LIN {X 0,Y 132.447,Z 765.257,A -85,B 0,C 180,E1 -26047.408,E2 -26047.408} C_VEL
LIN {X 0,Y 138.714,Z 760.063,A -85,B 0,C 180,E1 -26051.191,E2 -26051.191} C_VEL
LIN {X 0,Y 145.327,Z 753.801,A -85,B 0,C 180,E1 -26054.519,E2 -26054.519} C_VEL
LIN {X 0,Y 152.513,Z 746.044,A -85,B 0,C 180,E1 -26057.496,E2 -26057.496} C_VEL
LIN {X 0,Y 160.062,Z 736.576,A -85,B 0,C 180,E1 -26060.203,E2 -26060.203} C_VEL
LIN {X 0,Y 164.235,Z 730.683,A -85,B 0,C 180,E1 -26061.495,E2 -26061.495} C_VEL
LIN {X 0,Y 166.83,Z 726.274,A -85,B 0,C 180,E1 -26062.526,E2 -26062.526} C_VEL
LIN {X 0,Y 170.043,Z 719.082,A -85,B 0,C 180,E1 -26064.584,E2 -26064.584} C_VEL
LIN {X 0,Y 173.068,Z 711.529,A -85,B 0,C 180,E1 -26066.451,E2 -26066.451} C_VEL
LIN {X 0,Y 175.208,Z 706.525,A -85,B 0,C 180,E1 -26067.178,E2 -26067.178} C_VEL
LIN {X 0,Y 180.302,Z 693.883,A -85,B 0,C 180,E1 -26068.23,E2 -26068.23} C_VEL
LIN {X 0,Y 184.265,Z 680.937,A -85,B 0,C 180,E1 -26068.939,E2 -26068.939} C_VEL
LIN {X 0,Y 187.009,Z 667.101,A -85,B 0,C 180,E1 -26069.505,E2 -26069.505} C_VEL
LIN {X 0,Y 187.626,Z 662.527,A -85,B 0,C 180,E1 -26069.689,E2 -26069.689} C_VEL
LIN {X 0,Y 186.604,Z 658.475,A -85,B 0,C 180,E1 -26071.994,E2 -26071.994} C_VEL
LIN {X 0,Y 185.849,Z 655.332,A -85,B 0,C 180,E1 -26074.412,E2 -26074.412} C_VEL
LIN {X 0,Y 185.211,Z 652.435,A -85,B 0,C 180,E1 -26078.127,E2 -26078.127} C_VEL
LIN {X 0,Y 185.281,Z 651.918,A -85,B 0,C 180,E1 -26082.334,E2 -26082.334} C_VEL
LIN {X 0,Y 185.569,Z 652.744,A -85,B 0,C 180,E1 -26084.293,E2 -26084.293} C_VEL
LIN {X 0,Y 186.385,Z 654.34,A -85,B 0,C 180,E1 -26086.923,E2 -26086.923} C_VEL
LIN {X 0,Y 187.859,Z 658.008,A -85,B 0,C 180,E1 -26090.228,E2 -26090.228} C_VEL
LIN {X 0,Y 188.056,Z 658.81,A -85,B 0,C 180,E1 -26090.639,E2 -26090.639} C_VEL
LIN {X 0,Y 185.703,Z 673.409,A -85,B 0,C 180,E1 -26091.189,E2 -26091.189} C_VEL
LIN {X 0,Y 182.838,Z 684.634,A -85,B 0,C 180,E1 -26091.779,E2 -26091.779} C_VEL
LIN {X 0,Y 178.416,Z 697.436,A -85,B 0,C 180,E1 -26092.794,E2 -26092.794} C_VEL
LIN {X 0,Y 173.099,Z 709.329,A -85,B 0,C 180,E1 -26094.074,E2 -26094.074} C_VEL
LIN {X 0,Y 166.656,Z 720.747,A -85,B 0,C 180,E1 -26095.733,E2 -26095.733} C_VEL
LIN {X 0,Y 159.809,Z 730.899,A -85,B 0,C 180,E1 -26097.738,E2 -26097.738} C_VEL
LIN {X 0,Y 152.291,Z 740.223,A -85,B 0,C 180,E1 -26100.221,E2 -26100.221} C_VEL
LIN {X 0,Y 144.251,Z 748.58,A -85,B 0,C 180,E1 -26103.302,E2 -26103.302} C_VEL
LIN {X 0,Y 136.666,Z 755.296,A -85,B 0,C 180,E1 -26106.768,E2 -26106.768} C_VEL
LIN {X 0,Y 128.931,Z 761.128,A -85,B 0,C 180,E1 -26111.16,E2 -26111.16} C_VEL
LIN {X 0,Y 123.586,Z 764.553,A -85,B 0,C 180,E1 -26114.838,E2 -26114.838} C_VEL
LIN {X 0,Y 118.819,Z 767.124,A -85,B 0,C 180,E1 -26118.864,E2 -26118.864} C_VEL
LIN {X 0,Y 114.668,Z 768.928,A -85,B 0,C 180,E1 -26123.183,E2 -26123.183} C_VEL
LIN {X 0,Y 111.22,Z 770.025,A -85,B 0,C 180,E1 -26127.802,E2 -26127.802} C_VEL
LIN {X 0,Y 108.49,Z 770.374,A -85,B 0,C 180,E1 -26132.644,E2 -26132.644} C_VEL
LIN {X 0,Y 106.536,Z 770.012,A -85,B 0,C 180,E1 -26137.672,E2 -26137.672} C_VEL
LIN {X 0,Y 105.251,Z 768.99,A -85,B 0,C 180,E1 -26142.742,E2 -26142.742} C_VEL
LIN {X 0,Y 104.576,Z 766.125,A -85,B 0,C 180,E1 -26150.332,E2 -26150.332} C_VEL
LIN {X 0,Y 105.237,Z 761.777,A -85,B 0,C 180,E1 -26157.713,E2 -26157.713} C_VEL
LIN {X 0,Y 106.264,Z 757.954,A -85,B 0,C 180,E1 -26162.428,E2 -26162.428} C_VEL
LIN {X 0,Y 108.104,Z 752.178,A -85,B 0,C 180,E1 -26168.055,E2 -26168.055} C_VEL
LIN {X 0,Y 110.804,Z 744.691,A -85,B 0,C 180,E1 -26173.634,E2 -26173.634} C_VEL
LIN {X 0,Y 113.995,Z 736.372,A -85,B 0,C 180,E1 -26178.379,E2 -26178.379} C_VEL
LIN {X 0,Y 117.599,Z 726.557,A -85,B 0,C 180,E1 -26182.709,E2 -26182.709} C_VEL
LIN {X 0,Y 121.306,Z 715.813,A -85,B 0,C 180,E1 -26186.285,E2 -26186.285} C_VEL
LIN {X 0,Y 124.804,Z 704.272,A -85,B 0,C 180,E1 -26189.198,E2 -26189.198} C_VEL
LIN {X 0,Y 127.718,Z 692.806,A -85,B 0,C 180,E1 -26191.384,E2 -26191.384} C_VEL
LIN {X 0,Y 130.34,Z 679.686,A -85,B 0,C 180,E1 -26193.174,E2 -26193.174} C_VEL
LIN {X 0,Y 132.151,Z 667.516,A -85,B 0,C 180,E1 -26194.297,E2 -26194.297} C_VEL
LIN {X 0,Y 136.032,Z 623.336,A -85,B 0,C 180,E1 -26196.683,E2 -26196.683} C_VEL
LIN {X 0,Y 134.819,Z 619.141,A -85,B 0,C 180,E1 -26197.366,E2 -26197.366} C_VEL
LIN {X 0,Y 128.431,Z 604.449,A -85,B 0,C 180,E1 -26200.658,E2 -26200.658} C_VEL
LIN {X 0,Y 120.282,Z 590.115,A -85,B 0,C 180,E1 -26205.087,E2 -26205.087} C_VEL
LIN {X 0,Y 115.946,Z 583.556,A -85,B 0,C 180,E1 -26207.714,E2 -26207.714} C_VEL
LIN {X 0,Y 113.629,Z 580.152,A -85,B 0,C 180,E1 -26209.199,E2 -26209.199} C_VEL
LIN {X 0,Y 111.403,Z 576.9,A -85,B 0,C 180,E1 -26210.723,E2 -26210.723} C_VEL
LIN {X 0,Y 110.71,Z 575.798,A -85,B 0,C 180,E1 -26211.23,E2 -26211.23} C_VEL
LIN {X 0,Y 108.679,Z 573.458,A -85,B 0,C 180,E1 -26212.674,E2 -26212.674} C_VEL
LIN {X 0,Y 107.911,Z 571.002,A -85,B 0,C 180,E1 -26213.502,E2 -26213.502} C_VEL
LIN {X 0,Y 107.782,Z 571.046,A -85,B 0,C 180,E1 -26222.044,E2 -26222.044} C_VEL
LIN {X 0,Y 107.691,Z 571.063,A -85,B 0,C 180,E1 -26228.455,E2 -26228.455} C_VEL
LIN {X 0,Y 107.681,Z 571.072,A -85,B 0,C 180,E1 -26235.891,E2 -26235.891} C_VEL
LIN {X 0,Y 107.692,Z 571.048,A -85,B 0,C 180,E1 -26241.555,E2 -26241.555} C_VEL
LIN {X 0,Y 107.799,Z 571.045,A -85,B 0,C 180,E1 -26248.565,E2 -26248.565} C_VEL
LIN {X 0,Y 107.917,Z 571.042,A -85,B 0,C 180,E1 -26257.001,E2 -26257.001} C_VEL
LIN {X 0,Y 108.031,Z 571.01,A -85,B 0,C 180,E1 -26264.919,E2 -26264.919} C_VEL
LIN {X 0,Y 108.264,Z 570.998,A -85,B 0,C 180,E1 -26268.772,E2 -26268.772} C_VEL
LIN {X 0,Y 108.455,Z 570.964,A -85,B 0,C 180,E1 -26276.286,E2 -26276.286} C_VEL
LIN {X 0,Y 108.952,Z 570.912,A -85,B 0,C 180,E1 -26280.002,E2 -26280.002} C_VEL
LIN {X 0,Y 108.346,Z 570.987,A -85,B 0,C 180,E1 -26287.456,E2 -26287.456} C_VEL
LIN {X 0,Y 108.212,Z 570.989,A -85,B 0,C 180,E1 -26293.023,E2 -26293.023} C_VEL
LIN {X 0,Y 107.915,Z 571.036,A -85,B 0,C 180,E1 -26299.006,E2 -26299.006} C_VEL
LIN {X 0,Y 107.855,Z 571.003,A -85,B 0,C 180,E1 -26305.296,E2 -26305.296} C_VEL
LIN {X 0,Y 107.817,Z 571.013,A -85,B 0,C 180,E1 -26305.994,E2 -26305.994} C_VEL
LIN {X 0,Y 108.711,Z 573.751,A -85,B 0,C 180,E1 -26306.909,E2 -26306.909} C_VEL
LIN {X 0,Y 110.571,Z 575.854,A -85,B 0,C 180,E1 -26308.214,E2 -26308.214} C_VEL
LIN {X 0,Y 113.307,Z 579.959,A -85,B 0,C 180,E1 -26310.115,E2 -26310.115} C_VEL
LIN {X 0,Y 118.753,Z 588.444,A -85,B 0,C 180,E1 -26313.605,E2 -26313.605} C_VEL
LIN {X 0,Y 124.244,Z 597.99,A -85,B 0,C 180,E1 -26316.762,E2 -26316.762} C_VEL
LIN {X 0,Y 129.819,Z 611.769,A -85,B 0,C 180,E1 -26319.961,E2 -26319.961} C_VEL
LIN {X 0,Y 135.488,Z 628.741,A -85,B 0,C 180,E1 -26323.081,E2 -26323.081} C_VEL
LIN {X 0,Y 135.646,Z 631.726,A -85,B 0,C 180,E1 -26323.354,E2 -26323.354} C_VEL
LIN {X 0,Y 132.031,Z 673.668,A -85,B 0,C 180,E1 -26325.641,E2 -26325.641} C_VEL
LIN {X 0,Y 129.887,Z 687.418,A -85,B 0,C 180,E1 -26326.906,E2 -26326.906} C_VEL
LIN {X 0,Y 127.346,Z 699.278,A -85,B 0,C 180,E1 -26328.522,E2 -26328.522} C_VEL
LIN {X 0,Y 124.019,Z 711.744,A -85,B 0,C 180,E1 -26330.912,E2 -26330.912} C_VEL
LIN {X 0,Y 120.526,Z 722.973,A -85,B 0,C 180,E1 -26333.809,E2 -26333.809} C_VEL
LIN {X 0,Y 116.845,Z 733.399,A -85,B 0,C 180,E1 -26337.362,E2 -26337.362} C_VEL
LIN {X 0,Y 113.501,Z 742.302,A -85,B 0,C 180,E1 -26341.317,E2 -26341.317} C_VEL
LIN {X 0,Y 110.183,Z 751.263,A -85,B 0,C 180,E1 -26346.5,E2 -26346.5} C_VEL
LIN {X 0,Y 107.644,Z 758.393,A -85,B 0,C 180,E1 -26351.928,E2 -26351.928} C_VEL
LIN {X 0,Y 105.957,Z 764.887,A -85,B 0,C 180,E1 -26358.517,E2 -26358.517} C_VEL
